LIN {X 0,Y 334.452,Z 401.269,A -85,B 0,C 180,E1 -14668.793,E2 -14668.793} C_VEL
LIN {X 0,Y 334.325,Z 404.538,A -85,B 0,C 180,E1 -14671.202,E2 -14671.202} C_VEL
LIN {X 0,Y 333.817,Z 411.373,A -85,B 0,C 180,E1 -14676.04,E2 -14676.04} C_VEL
LIN {X 0,Y 333.325,Z 416.707,A -85,B 0,C 180,E1 -14679.708,E2 -14679.708} C_VEL
LIN {X 0,Y 332.922,Z 422.789,A -85,B 0,C 180,E1 -14683.819,E2 -14683.819} C_VEL
LIN {X 0,Y 332.746,Z 425.377,A -85,B 0,C 180,E1 -14685.541,E2 -14685.541} C_VEL
LIN {X 0,Y 335.286,Z 437.671,A -85,B 0,C 180,E1 -14686.278,E2 -14686.278} C_VEL
LIN {X 0,Y 337.14,Z 448.371,A -85,B 0,C 180,E1 -14687.121,E2 -14687.121} C_VEL
LIN {X 0,Y 337.706,Z 453.161,A -85,B 0,C 180,E1 -14687.56,E2 -14687.56} C_VEL
LIN {X 0,Y 336.838,Z 463.101,A -85,B 0,C 180,E1 -14688.55,E2 -14688.55} C_VEL
LIN {X 0,Y 335.882,Z 473.522,A -85,B 0,C 180,E1 -14689.887,E2 -14689.887} C_VEL
LIN {X 0,Y 335.116,Z 481.598,A -85,B 0,C 180,E1 -14691.205,E2 -14691.205} C_VEL
LIN {X 0,Y 334.312,Z 488.548,A -85,B 0,C 180,E1 -14692.594,E2 -14692.594} C_VEL
LIN {X 0,Y 333.638,Z 495.183,A -85,B 0,C 180,E1 -14694.249,E2 -14694.249} C_VEL
LIN {X 0,Y 332.933,Z 501.458,A -85,B 0,C 180,E1 -14696.311,E2 -14696.311} C_VEL
LIN {X 0,Y 332.49,Z 505.928,A -85,B 0,C 180,E1 -14698.394,E2 -14698.394} C_VEL
LIN {X 0,Y 332.162,Z 508.838,A -85,B 0,C 180,E1 -14700.513,E2 -14700.513} C_VEL
LIN {X 0,Y 332.04,Z 510.039,A -85,B 0,C 180,E1 -14702.152,E2 -14702.152} C_VEL
LIN {X 0,Y 332.048,Z 510.377,A -85,B 0,C 180,E1 -14703.384,E2 -14703.384} C_VEL
LIN {X 0,Y 332.14,Z 510.099,A -85,B 0,C 180,E1 -14704.838,E2 -14704.838} C_VEL
LIN {X 0,Y 332.357,Z 508.921,A -85,B 0,C 180,E1 -14706.531,E2 -14706.531} C_VEL
LIN {X 0,Y 332.817,Z 506.101,A -85,B 0,C 180,E1 -14708.619,E2 -14708.619} C_VEL
LIN {X 0,Y 333.451,Z 501.852,A -85,B 0,C 180,E1 -14710.646,E2 -14710.646} C_VEL
LIN {X 0,Y 334.247,Z 496.051,A -85,B 0,C 180,E1 -14712.615,E2 -14712.615} C_VEL
LIN {X 0,Y 335.069,Z 490.017,A -85,B 0,C 180,E1 -14714.188,E2 -14714.188} C_VEL
LIN {X 0,Y 336.238,Z 481.51,A -85,B 0,C 180,E1 -14715.923,E2 -14715.923} C_VEL
LIN {X 0,Y 337.346,Z 473.22,A -85,B 0,C 180,E1 -14717.249,E2 -14717.249} C_VEL
LIN {X 0,Y 338.217,Z 465.547,A -85,B 0,C 180,E1 -14718.255,E2 -14718.255} C_VEL
LIN {X 0,Y 338.19,Z 462.356,A -85,B 0,C 180,E1 -14718.645,E2 -14718.645} C_VEL
LIN {X 0,Y 337.525,Z 459.239,A -85,B 0,C 180,E1 -14719.042,E2 -14719.042} C_VEL
LIN {X 0,Y 335.005,Z 453.218,A -85,B 0,C 180,E1 -14719.825,E2 -14719.825} C_VEL
LIN {X 0,Y 331.983,Z 447.052,A -85,B 0,C 180,E1 -14720.571,E2 -14720.571} C_VEL
LIN {X 0,Y 330.188,Z 442.057,A -85,B 0,C 180,E1 -14721.074,E2 -14721.074} C_VEL
LIN {X 0,Y 329.772,Z 440.283,A -85,B 0,C 180,E1 -14721.225,E2 -14721.225} C_VEL
LIN {X 0,Y 326.593,Z 428.367,A -85,B 0,C 180,E1 -14722.124,E2 -14722.124} C_VEL
LIN {X 0,Y 326.223,Z 426.561,A -85,B 0,C 180,E1 -14722.269,E2 -14722.269} C_VEL
LIN {X 0,Y 326.561,Z 421.444,A -85,B 0,C 180,E1 -14725.976,E2 -14725.976} C_VEL
LIN {X 0,Y 326.992,Z 415.563,A -85,B 0,C 180,E1 -14730.375,E2 -14730.375} C_VEL
LIN {X 0,Y 327.403,Z 411.837,A -85,B 0,C 180,E1 -14733.206,E2 -14733.206} C_VEL
LIN {X 0,Y 327.616,Z 408.363,A -85,B 0,C 180,E1 -14735.947,E2 -14735.947} C_VEL
LIN {X 0,Y 327.526,Z 405.191,A -85,B 0,C 180,E1 -14738.606,E2 -14738.606} C_VEL
LIN {X 0,Y 327.156,Z 402.286,A -85,B 0,C 180,E1 -14741.203,E2 -14741.203} C_VEL
LIN {X 0,Y 326.68,Z 399.798,A -85,B 0,C 180,E1 -14743.599,E2 -14743.599} C_VEL
LIN {X 0,Y 326.741,Z 399.788,A -85,B 0,C 180,E1 -14746.314,E2 -14746.314} C_VEL
LIN {X 0,Y 326.793,Z 399.779,A -85,B 0,C 180,E1 -14750.094,E2 -14750.094} C_VEL
LIN {X 0,Y 326.958,Z 399.76,A -85,B 0,C 180,E1 -14752.59,E2 -14752.59} C_VEL
LIN {X 0,Y 326.767,Z 399.785,A -85,B 0,C 180,E1 -14755.065,E2 -14755.065} C_VEL
LIN {X 0,Y 327.056,Z 399.748,A -85,B 0,C 180,E1 -14757.537,E2 -14757.537} C_VEL
LIN {X 0,Y 327.216,Z 399.727,A -85,B 0,C 180,E1 -14760,E2 -14760} C_VEL
LIN {X 0,Y 327.056,Z 399.747,A -85,B 0,C 180,E1 -14762.464,E2 -14762.464} C_VEL
LIN {X 0,Y 326.978,Z 399.751,A -85,B 0,C 180,E1 -14766.17,E2 -14766.17} C_VEL
LIN {X 0,Y 326.893,Z 399.765,A -85,B 0,C 180,E1 -14768.656,E2 -14768.656} C_VEL
LIN {X 0,Y 326.718,Z 399.783,A -85,B 0,C 180,E1 -14772.422,E2 -14772.422} C_VEL
LIN {X 0,Y 326.733,Z 399.783,A -85,B 0,C 180,E1 -14774.959,E2 -14774.959} C_VEL
LIN {X 0,Y 326.716,Z 399.783,A -85,B 0,C 180,E1 -14778.842,E2 -14778.842} C_VEL
LIN {X 0,Y 326.624,Z 399.801,A -85,B 0,C 180,E1 -14782.788,E2 -14782.788} C_VEL
LIN {X 0,Y 326.673,Z 399.794,A -85,B 0,C 180,E1 -14785.486,E2 -14785.486} C_VEL
LIN {X 0,Y 326.643,Z 399.792,A -85,B 0,C 180,E1 -14789.661,E2 -14789.661} C_VEL
LIN {X 0,Y 326.59,Z 399.804,A -85,B 0,C 180,E1 -14794.022,E2 -14794.022} C_VEL
LIN {X 0,Y 326.613,Z 399.802,A -85,B 0,C 180,E1 -14797.242,E2 -14797.242} C_VEL
LIN {X 0,Y 326.62,Z 399.801,A -85,B 0,C 180,E1 -14800.205,E2 -14800.205} C_VEL
LIN {X 0,Y 326.644,Z 399.799,A -85,B 0,C 180,E1 -14803.512,E2 -14803.512} C_VEL
LIN {X 0,Y 326.702,Z 399.906,A -85,B 0,C 180,E1 -14804.862,E2 -14804.862} C_VEL
LIN {X 0,Y 327.773,Z 405.318,A -85,B 0,C 180,E1 -14808.631,E2 -14808.631} C_VEL
LIN {X 0,Y 328.717,Z 410.195,A -85,B 0,C 180,E1 -14811.687,E2 -14811.687} C_VEL
LIN {X 0,Y 330.049,Z 416.95,A -85,B 0,C 180,E1 -14815.573,E2 -14815.573} C_VEL
LIN {X 0,Y 330.66,Z 421.324,A -85,B 0,C 180,E1 -14817.907,E2 -14817.907} C_VEL
LIN {X 0,Y 329.991,Z 425.615,A -85,B 0,C 180,E1 -14819.971,E2 -14819.971} C_VEL
LIN {X 0,Y 328.501,Z 434.354,A -85,B 0,C 180,E1 -14823.969,E2 -14823.969} C_VEL
LIN {X 0,Y 327.223,Z 443.457,A -85,B 0,C 180,E1 -14827.993,E2 -14827.993} C_VEL
LIN {X 0,Y 330.129,Z 458.426,A -85,B 0,C 180,E1 -14828.837,E2 -14828.837} C_VEL
LIN {X 0,Y 331.601,Z 471.167,A -85,B 0,C 180,E1 -14829.742,E2 -14829.742} C_VEL
LIN {X 0,Y 332.114,Z 482.072,A -85,B 0,C 180,E1 -14830.695,E2 -14830.695} C_VEL
LIN {X 0,Y 331.005,Z 492.541,A -85,B 0,C 180,E1 -14831.753,E2 -14831.753} C_VEL
LIN {X 0,Y 329.552,Z 503.242,A -85,B 0,C 180,E1 -14833.111,E2 -14833.111} C_VEL
LIN {X 0,Y 328.483,Z 512.049,A -85,B 0,C 180,E1 -14834.507,E2 -14834.507} C_VEL
LIN {X 0,Y 327.513,Z 519.964,A -85,B 0,C 180,E1 -14836.033,E2 -14836.033} C_VEL
LIN {X 0,Y 326.413,Z 527.732,A -85,B 0,C 180,E1 -14837.885,E2 -14837.885} C_VEL
LIN {X 0,Y 325.459,Z 536.929,A -85,B 0,C 180,E1 -14840.683,E2 -14840.683} C_VEL
LIN {X 0,Y 325.106,Z 542.054,A -85,B 0,C 180,E1 -14842.55,E2 -14842.55} C_VEL
LIN {X 0,Y 324.911,Z 545.74,A -85,B 0,C 180,E1 -14844.274,E2 -14844.274} C_VEL
LIN {X 0,Y 324.917,Z 548.848,A -85,B 0,C 180,E1 -14846.282,E2 -14846.282} C_VEL
LIN {X 0,Y 324.882,Z 550.174,A -85,B 0,C 180,E1 -14847.523,E2 -14847.523} C_VEL
LIN {X 0,Y 324.897,Z 551.09,A -85,B 0,C 180,E1 -14848.763,E2 -14848.763} C_VEL
LIN {X 0,Y 324.91,Z 551.588,A -85,B 0,C 180,E1 -14850.003,E2 -14850.003} C_VEL
LIN {X 0,Y 324.885,Z 551.632,A -85,B 0,C 180,E1 -14851.242,E2 -14851.242} C_VEL
LIN {X 0,Y 324.884,Z 551.275,A -85,B 0,C 180,E1 -14852.482,E2 -14852.482} C_VEL
LIN {X 0,Y 324.917,Z 550.521,A -85,B 0,C 180,E1 -14853.723,E2 -14853.723} C_VEL
LIN {X 0,Y 324.92,Z 548.385,A -85,B 0,C 180,E1 -14855.741,E2 -14855.741} C_VEL
LIN {X 0,Y 325.191,Z 545.655,A -85,B 0,C 180,E1 -14857.453,E2 -14857.453} C_VEL
LIN {X 0,Y 325.607,Z 541.696,A -85,B 0,C 180,E1 -14859.319,E2 -14859.319} C_VEL
LIN {X 0,Y 326.431,Z 535.61,A -85,B 0,C 180,E1 -14861.49,E2 -14861.49} C_VEL
LIN {X 0,Y 327.445,Z 528.982,A -85,B 0,C 180,E1 -14863.342,E2 -14863.342} C_VEL
LIN {X 0,Y 328.79,Z 520.814,A -85,B 0,C 180,E1 -14865.182,E2 -14865.182} C_VEL
LIN {X 0,Y 329.975,Z 512.524,A -85,B 0,C 180,E1 -14866.712,E2 -14866.712} C_VEL
LIN {X 0,Y 331.648,Z 502.355,A -85,B 0,C 180,E1 -14868.216,E2 -14868.216} C_VEL
LIN {X 0,Y 333.175,Z 492.443,A -85,B 0,C 180,E1 -14869.407,E2 -14869.407} C_VEL
LIN {X 0,Y 334.141,Z 483.521,A -85,B 0,C 180,E1 -14870.309,E2 -14870.309} C_VEL
LIN {X 0,Y 333.854,Z 472.11,A -85,B 0,C 180,E1 -14871.365,E2 -14871.365} C_VEL
LIN {X 0,Y 332.316,Z 458.96,A -85,B 0,C 180,E1 -14872.419,E2 -14872.419} C_VEL
LIN {X 0,Y 329.655,Z 445.962,A -85,B 0,C 180,E1 -14873.306,E2 -14873.306} C_VEL
LIN {X 0,Y 327.517,Z 437.12,A -85,B 0,C 180,E1 -14873.863,E2 -14873.863} C_VEL
LIN {X 0,Y 328.673,Z 429.043,A -85,B 0,C 180,E1 -14877.372,E2 -14877.372} C_VEL
LIN {X 0,Y 329.908,Z 421.406,A -85,B 0,C 180,E1 -14880.751,E2 -14880.751} C_VEL
LIN {X 0,Y 330.137,Z 418.339,A -85,B 0,C 180,E1 -14882.157,E2 -14882.157} C_VEL
LIN {X 0,Y 329.022,Z 412.165,A -85,B 0,C 180,E1 -14885.223,E2 -14885.223} C_VEL
LIN {X 0,Y 327.48,Z 404.167,A -85,B 0,C 180,E1 -14889.412,E2 -14889.412} C_VEL
LIN {X 0,Y 326.602,Z 399.803,A -85,B 0,C 180,E1 -14891.844,E2 -14891.844} C_VEL
LIN {X 0,Y 326.532,Z 399.81,A -85,B 0,C 180,E1 -14895.259,E2 -14895.259} C_VEL
LIN {X 0,Y 326.569,Z 399.805,A -85,B 0,C 180,E1 -14898.153,E2 -14898.153} C_VEL
LIN {X 0,Y 326.59,Z 399.798,A -85,B 0,C 180,E1 -14901.386,E2 -14901.386} C_VEL
LIN {X 0,Y 326.627,Z 399.8,A -85,B 0,C 180,E1 -14904.852,E2 -14904.852} C_VEL
LIN {X 0,Y 326.616,Z 399.8,A -85,B 0,C 180,E1 -14907.456,E2 -14907.456} C_VEL
LIN {X 0,Y 326.597,Z 399.802,A -85,B 0,C 180,E1 -14910.334,E2 -14910.334} C_VEL
LIN {X 0,Y 326.603,Z 399.802,A -85,B 0,C 180,E1 -14913.135,E2 -14913.135} C_VEL
LIN {X 0,Y 326.598,Z 399.803,A -85,B 0,C 180,E1 -14917.211,E2 -14917.211} C_VEL
LIN {X 0,Y 326.754,Z 399.784,A -85,B 0,C 180,E1 -14921.178,E2 -14921.178} C_VEL
LIN {X 0,Y 326.772,Z 399.784,A -85,B 0,C 180,E1 -14925.433,E2 -14925.433} C_VEL
LIN {X 0,Y 326.788,Z 399.871,A -85,B 0,C 180,E1 -14929.545,E2 -14929.545} C_VEL
LIN {X 0,Y 327.805,Z 404.409,A -85,B 0,C 180,E1 -14932.609,E2 -14932.609} C_VEL
LIN {X 0,Y 328.363,Z 408.303,A -85,B 0,C 180,E1 -14935.088,E2 -14935.088} C_VEL
LIN {X 0,Y 328.368,Z 412.44,A -85,B 0,C 180,E1 -14937.546,E2 -14937.546} C_VEL
LIN {X 0,Y 327.807,Z 417.739,A -85,B 0,C 180,E1 -14940.614,E2 -14940.614} C_VEL
LIN {X 0,Y 327.262,Z 425.21,A -85,B 0,C 180,E1 -14944.927,E2 -14944.927} C_VEL
LIN {X 0,Y 327.074,Z 428.969,A -85,B 0,C 180,E1 -14947.097,E2 -14947.097} C_VEL
LIN {X 0,Y 331.673,Z 443.489,A -85,B 0,C 180,E1 -14948.319,E2 -14948.319} C_VEL
LIN {X 0,Y 334.363,Z 455.286,A -85,B 0,C 180,E1 -14949.406,E2 -14949.406} C_VEL
LIN {X 0,Y 335.716,Z 465.144,A -85,B 0,C 180,E1 -14950.402,E2 -14950.402} C_VEL
LIN {X 0,Y 334.254,Z 476.454,A -85,B 0,C 180,E1 -14951.522,E2 -14951.522} C_VEL
LIN {X 0,Y 332.591,Z 487.852,A -85,B 0,C 180,E1 -14952.949,E2 -14952.949} C_VEL
LIN {X 0,Y 331.025,Z 497.442,A -85,B 0,C 180,E1 -14954.445,E2 -14954.445} C_VEL
LIN {X 0,Y 329.425,Z 506.719,A -85,B 0,C 180,E1 -14956.248,E2 -14956.248} C_VEL
LIN {X 0,Y 328.113,Z 514.369,A -85,B 0,C 180,E1 -14958.094,E2 -14958.094} C_VEL
LIN {X 0,Y 326.984,Z 520.949,A -85,B 0,C 180,E1 -14960.114,E2 -14960.114} C_VEL
LIN {X 0,Y 326.086,Z 525.896,A -85,B 0,C 180,E1 -14962.061,E2 -14962.061} C_VEL
LIN {X 0,Y 325.474,Z 529.964,A -85,B 0,C 180,E1 -14964.221,E2 -14964.221} C_VEL
LIN {X 0,Y 325.17,Z 531.838,A -85,B 0,C 180,E1 -14965.611,E2 -14965.611} C_VEL
LIN {X 0,Y 324.841,Z 533.562,A -85,B 0,C 180,E1 -14967.493,E2 -14967.493} C_VEL
LIN {X 0,Y 324.622,Z 534.411,A -85,B 0,C 180,E1 -14970.001,E2 -14970.001} C_VEL
LIN {X 0,Y 324.582,Z 533.648,A -85,B 0,C 180,E1 -14972.385,E2 -14972.385} C_VEL
LIN {X 0,Y 324.76,Z 531.489,A -85,B 0,C 180,E1 -14974.677,E2 -14974.677} C_VEL
LIN {X 0,Y 325.157,Z 528.008,A -85,B 0,C 180,E1 -14976.894,E2 -14976.894} C_VEL
LIN {X 0,Y 325.542,Z 523.285,A -85,B 0,C 180,E1 -14978.993,E2 -14978.993} C_VEL
LIN {X 0,Y 326.14,Z 517.232,A -85,B 0,C 180,E1 -14981.041,E2 -14981.041} C_VEL
LIN {X 0,Y 326.915,Z 509.69,A -85,B 0,C 180,E1 -14983.033,E2 -14983.033} C_VEL
LIN {X 0,Y 327.913,Z 500.349,A -85,B 0,C 180,E1 -14984.984,E2 -14984.984} C_VEL
LIN {X 0,Y 329.014,Z 490.812,A -85,B 0,C 180,E1 -14986.574,E2 -14986.574} C_VEL
LIN {X 0,Y 330.099,Z 480.41,A -85,B 0,C 180,E1 -14987.98,E2 -14987.98} C_VEL
LIN {X 0,Y 331.204,Z 469.031,A -85,B 0,C 180,E1 -14989.216,E2 -14989.216} C_VEL
LIN {X 0,Y 331.864,Z 460.882,A -85,B 0,C 180,E1 -14989.933,E2 -14989.933} C_VEL
LIN {X 0,Y 330.017,Z 448.543,A -85,B 0,C 180,E1 -14990.934,E2 -14990.934} C_VEL
LIN {X 0,Y 327.287,Z 434.324,A -85,B 0,C 180,E1 -14991.825,E2 -14991.825} C_VEL
LIN {X 0,Y 325.942,Z 427.724,A -85,B 0,C 180,E1 -14992.178,E2 -14992.178} C_VEL
LIN {X 0,Y 326.253,Z 420.978,A -85,B 0,C 180,E1 -14995.936,E2 -14995.936} C_VEL
LIN {X 0,Y 326.542,Z 414.759,A -85,B 0,C 180,E1 -14999.417,E2 -14999.417} C_VEL
LIN {X 0,Y 326.776,Z 409.236,A -85,B 0,C 180,E1 -15002.507,E2 -15002.507} C_VEL
LIN {X 0,Y 327.051,Z 403.236,A -85,B 0,C 180,E1 -15005.9,E2 -15005.9} C_VEL
LIN {X 0,Y 326.775,Z 399.782,A -85,B 0,C 180,E1 -15007.93,E2 -15007.93} C_VEL
LIN {X 0,Y 326.747,Z 399.785,A -85,B 0,C 180,E1 -15011.175,E2 -15011.175} C_VEL
LIN {X 0,Y 326.765,Z 399.784,A -85,B 0,C 180,E1 -15015.431,E2 -15015.431} C_VEL
LIN {X 0,Y 326.771,Z 399.782,A -85,B 0,C 180,E1 -15018.836,E2 -15018.836} C_VEL
LIN {X 0,Y 326.923,Z 399.764,A -85,B 0,C 180,E1 -15022.587,E2 -15022.587} C_VEL
LIN {X 0,Y 326.754,Z 399.789,A -85,B 0,C 180,E1 -15025.062,E2 -15025.062} C_VEL
LIN {X 0,Y 326.832,Z 399.839,A -85,B 0,C 180,E1 -15026.761,E2 -15026.761} C_VEL
LIN {X 0,Y 327.447,Z 402.365,A -85,B 0,C 180,E1 -15028.767,E2 -15028.767} C_VEL
LIN {X 0,Y 327.295,Z 405.666,A -85,B 0,C 180,E1 -15031.228,E2 -15031.228} C_VEL
LIN {X 0,Y 326.744,Z 412.542,A -85,B 0,C 180,E1 -15036.171,E2 -15036.171} C_VEL
LIN {X 0,Y 326.262,Z 417.889,A -85,B 0,C 180,E1 -15039.92,E2 -15039.92} C_VEL
LIN {X 0,Y 325.847,Z 423.753,A -85,B 0,C 180,E1 -15043.935,E2 -15043.935} C_VEL
LIN {X 0,Y 325.743,Z 425.557,A -85,B 0,C 180,E1 -15045.162,E2 -15045.162} C_VEL
LIN {X 0,Y 328.436,Z 438.699,A -85,B 0,C 180,E1 -15045.989,E2 -15045.989} C_VEL
LIN {X 0,Y 330.221,Z 449.282,A -85,B 0,C 180,E1 -15046.853,E2 -15046.853} C_VEL
LIN {X 0,Y 330.806,Z 453.971,A -85,B 0,C 180,E1 -15047.3,E2 -15047.3} C_VEL
LIN {X 0,Y 329.915,Z 463.778,A -85,B 0,C 180,E1 -15048.31,E2 -15048.31} C_VEL
LIN {X 0,Y 328.986,Z 473.555,A -85,B 0,C 180,E1 -15049.59,E2 -15049.59} C_VEL
LIN {X 0,Y 328.119,Z 482.163,A -85,B 0,C 180,E1 -15051.021,E2 -15051.021} C_VEL
LIN {X 0,Y 327.137,Z 490.412,A -85,B 0,C 180,E1 -15052.746,E2 -15052.746} C_VEL
LIN {X 0,Y 326.37,Z 497.455,A -85,B 0,C 180,E1 -15054.663,E2 -15054.663} C_VEL
LIN {X 0,Y 325.87,Z 501.929,A -85,B 0,C 180,E1 -15056.236,E2 -15056.236} C_VEL
LIN {X 0,Y 325.414,Z 506.379,A -85,B 0,C 180,E1 -15058.364,E2 -15058.364} C_VEL
LIN {X 0,Y 325.128,Z 508.903,A -85,B 0,C 180,E1 -15060.159,E2 -15060.159} C_VEL
LIN {X 0,Y 325.001,Z 509.9,A -85,B 0,C 180,E1 -15061.26,E2 -15061.26} C_VEL
LIN {X 0,Y 324.963,Z 510.663,A -85,B 0,C 180,E1 -15062.726,E2 -15062.726} C_VEL
LIN {X 0,Y 325.051,Z 510.568,A -85,B 0,C 180,E1 -15064.755,E2 -15064.755} C_VEL
LIN {X 0,Y 325.356,Z 509.042,A -85,B 0,C 180,E1 -15066.944,E2 -15066.944} C_VEL
LIN {X 0,Y 325.893,Z 506.035,A -85,B 0,C 180,E1 -15069.073,E2 -15069.073} C_VEL
LIN {X 0,Y 326.539,Z 501.602,A -85,B 0,C 180,E1 -15071.124,E2 -15071.124} C_VEL
LIN {X 0,Y 327.443,Z 495.596,A -85,B 0,C 180,E1 -15073.135,E2 -15073.135} C_VEL
LIN {X 0,Y 328.451,Z 488.585,A -85,B 0,C 180,E1 -15074.914,E2 -15074.914} C_VEL
LIN {X 0,Y 329.56,Z 480.771,A -85,B 0,C 180,E1 -15076.469,E2 -15076.469} C_VEL
LIN {X 0,Y 330.919,Z 470.893,A -85,B 0,C 180,E1 -15078.01,E2 -15078.01} C_VEL
LIN {X 0,Y 332.054,Z 461.076,A -85,B 0,C 180,E1 -15079.202,E2 -15079.202} C_VEL
LIN {X 0,Y 332.497,Z 456.981,A -85,B 0,C 180,E1 -15079.619,E2 -15079.619} C_VEL
LIN {X 0,Y 331.184,Z 447.065,A -85,B 0,C 180,E1 -15080.627,E2 -15080.627} C_VEL
LIN {X 0,Y 329.772,Z 440.283,A -85,B 0,C 180,E1 -15081.225,E2 -15081.225} C_VEL
LIN {X 0,Y 328.516,Z 438.347,A -85,B 0,C 180,E1 -15081.451,E2 -15081.451} C_VEL
LIN {X 0,Y 322.469,Z 435.25,A -85,B 0,C 180,E1 -15082.111,E2 -15082.111} C_VEL
LIN {X 0,Y 321.128,Z 433.6,A -85,B 0,C 180,E1 -15082.304,E2 -15082.304} C_VEL
LIN {X 0,Y 319.257,Z 426.842,A -85,B 0,C 180,E1 -15082.787,E2 -15082.787} C_VEL
LIN {X 0,Y 319.608,Z 421.628,A -85,B 0,C 180,E1 -15086.671,E2 -15086.671} C_VEL
LIN {X 0,Y 319.882,Z 417.736,A -85,B 0,C 180,E1 -15089.648,E2 -15089.648} C_VEL
LIN {X 0,Y 320.324,Z 413.962,A -85,B 0,C 180,E1 -15092.565,E2 -15092.565} C_VEL
LIN {X 0,Y 320.608,Z 410.436,A -85,B 0,C 180,E1 -15095.387,E2 -15095.387} C_VEL
LIN {X 0,Y 320.602,Z 407.183,A -85,B 0,C 180,E1 -15098.121,E2 -15098.121} C_VEL
LIN {X 0,Y 320.283,Z 404.248,A -85,B 0,C 180,E1 -15100.783,E2 -15100.783} C_VEL
LIN {X 0,Y 319.672,Z 400.67,A -85,B 0,C 180,E1 -15104.377,E2 -15104.377} C_VEL
LIN {X 0,Y 319.664,Z 400.667,A -85,B 0,C 180,E1 -15107.3,E2 -15107.3} C_VEL
LIN {X 0,Y 319.859,Z 400.644,A -85,B 0,C 180,E1 -15111.369,E2 -15111.369} C_VEL
LIN {X 0,Y 319.932,Z 400.633,A -85,B 0,C 180,E1 -15113.695,E2 -15113.695} C_VEL
LIN {X 0,Y 319.996,Z 400.627,A -85,B 0,C 180,E1 -15117.483,E2 -15117.483} C_VEL
LIN {X 0,Y 320.167,Z 400.605,A -85,B 0,C 180,E1 -15120,E2 -15120} C_VEL
LIN {X 0,Y 319.996,Z 400.626,A -85,B 0,C 180,E1 -15122.518,E2 -15122.518} C_VEL
LIN {X 0,Y 319.933,Z 400.628,A -85,B 0,C 180,E1 -15126.306,E2 -15126.306} C_VEL
LIN {X 0,Y 319.821,Z 400.645,A -85,B 0,C 180,E1 -15128.849,E2 -15128.849} C_VEL
LIN {X 0,Y 319.664,Z 400.661,A -85,B 0,C 180,E1 -15132.701,E2 -15132.701} C_VEL
LIN {X 0,Y 319.679,Z 400.66,A -85,B 0,C 180,E1 -15135.297,E2 -15135.297} C_VEL
LIN {X 0,Y 319.66,Z 400.664,A -85,B 0,C 180,E1 -15139.256,E2 -15139.256} C_VEL
LIN {X 0,Y 319.566,Z 400.679,A -85,B 0,C 180,E1 -15143.32,E2 -15143.32} C_VEL
LIN {X 0,Y 319.617,Z 400.672,A -85,B 0,C 180,E1 -15146.09,E2 -15146.09} C_VEL
LIN {X 0,Y 319.571,Z 400.676,A -85,B 0,C 180,E1 -15148.936,E2 -15148.936} C_VEL
LIN {X 0,Y 319.515,Z 400.681,A -85,B 0,C 180,E1 -15151.864,E2 -15151.864} C_VEL
LIN {X 0,Y 319.563,Z 400.679,A -85,B 0,C 180,E1 -15155.546,E2 -15155.546} C_VEL
LIN {X 0,Y 319.584,Z 400.677,A -85,B 0,C 180,E1 -15158.007,E2 -15158.007} C_VEL
LIN {X 0,Y 319.587,Z 400.678,A -85,B 0,C 180,E1 -15161.615,E2 -15161.615} C_VEL
LIN {X 0,Y 319.629,Z 400.846,A -85,B 0,C 180,E1 -15164.042,E2 -15164.042} C_VEL
LIN {X 0,Y 320.545,Z 405.112,A -85,B 0,C 180,E1 -15167.187,E2 -15167.187} C_VEL
LIN {X 0,Y 321.557,Z 410.35,A -85,B 0,C 180,E1 -15170.672,E2 -15170.672} C_VEL
LIN {X 0,Y 322.851,Z 417.144,A -85,B 0,C 180,E1 -15174.774,E2 -15174.774} C_VEL
LIN {X 0,Y 323.599,Z 421.346,A -85,B 0,C 180,E1 -15177.119,E2 -15177.119} C_VEL
LIN {X 0,Y 323.545,Z 424.16,A -85,B 0,C 180,E1 -15178.583,E2 -15178.583} C_VEL
LIN {X 0,Y 321.886,Z 432.837,A -85,B 0,C 180,E1 -15182.713,E2 -15182.713} C_VEL
LIN {X 0,Y 320.53,Z 441.69,A -85,B 0,C 180,E1 -15186.758,E2 -15186.758} C_VEL
LIN {X 0,Y 320.32,Z 443.398,A -85,B 0,C 180,E1 -15187.485,E2 -15187.485} C_VEL
LIN {X 0,Y 322.976,Z 456.392,A -85,B 0,C 180,E1 -15188.214,E2 -15188.214} C_VEL
LIN {X 0,Y 324.618,Z 468.94,A -85,B 0,C 180,E1 -15189.111,E2 -15189.111} C_VEL
LIN {X 0,Y 325.293,Z 480.354,A -85,B 0,C 180,E1 -15190.109,E2 -15190.109} C_VEL
LIN {X 0,Y 325.034,Z 486.85,A -85,B 0,C 180,E1 -15190.75,E2 -15190.75} C_VEL
LIN {X 0,Y 323.571,Z 497.51,A -85,B 0,C 180,E1 -15191.974,E2 -15191.974} C_VEL
LIN {X 0,Y 322.031,Z 508.166,A -85,B 0,C 180,E1 -15193.521,E2 -15193.521} C_VEL
LIN {X 0,Y 320.935,Z 516.769,A -85,B 0,C 180,E1 -15195.093,E2 -15195.093} C_VEL
LIN {X 0,Y 319.848,Z 525.08,A -85,B 0,C 180,E1 -15196.987,E2 -15196.987} C_VEL
LIN {X 0,Y 318.966,Z 530.728,A -85,B 0,C 180,E1 -15198.565,E2 -15198.565} C_VEL
LIN {X 0,Y 318.154,Z 539.994,A -85,B 0,C 180,E1 -15201.748,E2 -15201.748} C_VEL
LIN {X 0,Y 317.889,Z 544.379,A -85,B 0,C 180,E1 -15203.656,E2 -15203.656} C_VEL
LIN {X 0,Y 317.814,Z 546.681,A -85,B 0,C 180,E1 -15204.928,E2 -15204.928} C_VEL
LIN {X 0,Y 317.823,Z 548.525,A -85,B 0,C 180,E1 -15206.199,E2 -15206.199} C_VEL
LIN {X 0,Y 317.801,Z 549.88,A -85,B 0,C 180,E1 -15207.468,E2 -15207.468} C_VEL
LIN {X 0,Y 317.805,Z 550.824,A -85,B 0,C 180,E1 -15208.736,E2 -15208.736} C_VEL
LIN {X 0,Y 317.816,Z 551.364,A -85,B 0,C 180,E1 -15210.003,E2 -15210.003} C_VEL
LIN {X 0,Y 317.794,Z 551.45,A -85,B 0,C 180,E1 -15211.27,E2 -15211.27} C_VEL
LIN {X 0,Y 317.802,Z 551.12,A -85,B 0,C 180,E1 -15212.538,E2 -15212.538} C_VEL
LIN {X 0,Y 317.823,Z 550.391,A -85,B 0,C 180,E1 -15213.806,E2 -15213.806} C_VEL
LIN {X 0,Y 317.838,Z 548.503,A -85,B 0,C 180,E1 -15215.707,E2 -15215.707} C_VEL
LIN {X 0,Y 318.13,Z 545.63,A -85,B 0,C 180,E1 -15217.62,E2 -15217.62} C_VEL
LIN {X 0,Y 318.588,Z 541.745,A -85,B 0,C 180,E1 -15219.526,E2 -15219.526} C_VEL
LIN {X 0,Y 319.321,Z 536.731,A -85,B 0,C 180,E1 -15221.427,E2 -15221.427} C_VEL
LIN {X 0,Y 320.305,Z 530.452,A -85,B 0,C 180,E1 -15223.322,E2 -15223.322} C_VEL
LIN {X 0,Y 321.718,Z 522.637,A -85,B 0,C 180,E1 -15225.2,E2 -15225.2} C_VEL
LIN {X 0,Y 323.194,Z 512.985,A -85,B 0,C 180,E1 -15227.073,E2 -15227.073} C_VEL
LIN {X 0,Y 324.951,Z 503.049,A -85,B 0,C 180,E1 -15228.606,E2 -15228.606} C_VEL
LIN {X 0,Y 326.55,Z 493.382,A -85,B 0,C 180,E1 -15229.817,E2 -15229.817} C_VEL
LIN {X 0,Y 327.62,Z 484.775,A -85,B 0,C 180,E1 -15230.732,E2 -15230.732} C_VEL
LIN {X 0,Y 327.406,Z 473.351,A -85,B 0,C 180,E1 -15231.84,E2 -15231.84} C_VEL
LIN {X 0,Y 326.036,Z 460.605,A -85,B 0,C 180,E1 -15232.917,E2 -15232.917} C_VEL
LIN {X 0,Y 323.471,Z 447.178,A -85,B 0,C 180,E1 -15233.903,E2 -15233.903} C_VEL
LIN {X 0,Y 320.742,Z 436.804,A -85,B 0,C 180,E1 -15234.605,E2 -15234.605} C_VEL
LIN {X 0,Y 320.705,Z 436.092,A -85,B 0,C 180,E1 -15234.694,E2 -15234.694} C_VEL
LIN {X 0,Y 322.082,Z 427.151,A -85,B 0,C 180,E1 -15238.691,E2 -15238.691} C_VEL
LIN {X 0,Y 323.061,Z 421.055,A -85,B 0,C 180,E1 -15241.476,E2 -15241.476} C_VEL
LIN {X 0,Y 322.908,Z 417.996,A -85,B 0,C 180,E1 -15242.967,E2 -15242.967} C_VEL
LIN {X 0,Y 321.703,Z 411.78,A -85,B 0,C 180,E1 -15246.149,E2 -15246.149} C_VEL
LIN {X 0,Y 320.405,Z 404.942,A -85,B 0,C 180,E1 -15249.85,E2 -15249.85} C_VEL
LIN {X 0,Y 319.543,Z 400.684,A -85,B 0,C 180,E1 -15252.347,E2 -15252.347} C_VEL
LIN {X 0,Y 319.526,Z 400.677,A -85,B 0,C 180,E1 -15256.541,E2 -15256.541} C_VEL
LIN {X 0,Y 319.553,Z 400.679,A -85,B 0,C 180,E1 -15260.371,E2 -15260.371} C_VEL
LIN {X 0,Y 319.587,Z 400.675,A -85,B 0,C 180,E1 -15264.458,E2 -15264.458} C_VEL
LIN {X 0,Y 319.532,Z 400.684,A -85,B 0,C 180,E1 -15268.138,E2 -15268.138} C_VEL
LIN {X 0,Y 319.575,Z 400.678,A -85,B 0,C 180,E1 -15271.606,E2 -15271.606} C_VEL
LIN {X 0,Y 319.534,Z 400.685,A -85,B 0,C 180,E1 -15275.298,E2 -15275.298} C_VEL
LIN {X 0,Y 319.573,Z 400.679,A -85,B 0,C 180,E1 -15278.046,E2 -15278.046} C_VEL
LIN {X 0,Y 319.698,Z 400.663,A -85,B 0,C 180,E1 -15280.963,E2 -15280.963} C_VEL
LIN {X 0,Y 319.74,Z 400.661,A -85,B 0,C 180,E1 -15285.276,E2 -15285.276} C_VEL
LIN {X 0,Y 319.721,Z 400.777,A -85,B 0,C 180,E1 -15288.589,E2 -15288.589} C_VEL
LIN {X 0,Y 320.589,Z 404.376,A -85,B 0,C 180,E1 -15291.172,E2 -15291.172} C_VEL
LIN {X 0,Y 321.305,Z 408.134,A -85,B 0,C 180,E1 -15293.721,E2 -15293.721} C_VEL
LIN {X 0,Y 321.59,Z 412.111,A -85,B 0,C 180,E1 -15296.24,E2 -15296.24} C_VEL
LIN {X 0,Y 321.307,Z 416.287,A -85,B 0,C 180,E1 -15298.746,E2 -15298.746} C_VEL
LIN {X 0,Y 320.454,Z 424.812,A -85,B 0,C 180,E1 -15303.772,E2 -15303.772} C_VEL
LIN {X 0,Y 320.229,Z 429.416,A -85,B 0,C 180,E1 -15306.379,E2 -15306.379} C_VEL
LIN {X 0,Y 324.781,Z 443.108,A -85,B 0,C 180,E1 -15307.589,E2 -15307.589} C_VEL
LIN {X 0,Y 327.728,Z 455.554,A -85,B 0,C 180,E1 -15308.788,E2 -15308.788} C_VEL
LIN {X 0,Y 329.115,Z 465.432,A -85,B 0,C 180,E1 -15309.836,E2 -15309.836} C_VEL
LIN {X 0,Y 328.513,Z 471.861,A -85,B 0,C 180,E1 -15310.476,E2 -15310.476} C_VEL
LIN {X 0,Y 326.819,Z 483.251,A -85,B 0,C 180,E1 -15311.788,E2 -15311.788} C_VEL
LIN {X 0,Y 325.063,Z 494.055,A -85,B 0,C 180,E1 -15313.359,E2 -15313.359} C_VEL
LIN {X 0,Y 323.281,Z 503.738,A -85,B 0,C 180,E1 -15315.122,E2 -15315.122} C_VEL
LIN {X 0,Y 321.98,Z 511.203,A -85,B 0,C 180,E1 -15316.81,E2 -15316.81} C_VEL
LIN {X 0,Y 320.574,Z 518.488,A -85,B 0,C 180,E1 -15318.866,E2 -15318.866} C_VEL
LIN {X 0,Y 319.676,Z 523.384,A -85,B 0,C 180,E1 -15320.594,E2 -15320.594} C_VEL
LIN {X 0,Y 318.789,Z 528.137,A -85,B 0,C 180,E1 -15322.763,E2 -15322.763} C_VEL
LIN {X 0,Y 318.202,Z 531.736,A -85,B 0,C 180,E1 -15325.099,E2 -15325.099} C_VEL
LIN {X 0,Y 317.941,Z 532.939,A -85,B 0,C 180,E1 -15326.237,E2 -15326.237} C_VEL
LIN {X 0,Y 317.7,Z 534.043,A -85,B 0,C 180,E1 -15327.762,E2 -15327.762} C_VEL
LIN {X 0,Y 317.555,Z 534.542,A -85,B 0,C 180,E1 -15329.136,E2 -15329.136} C_VEL
LIN {X 0,Y 317.489,Z 534.526,A -85,B 0,C 180,E1 -15330.606,E2 -15330.606} C_VEL
LIN {X 0,Y 317.498,Z 533.561,A -85,B 0,C 180,E1 -15332.735,E2 -15332.735} C_VEL
LIN {X 0,Y 317.741,Z 531.109,A -85,B 0,C 180,E1 -15335.105,E2 -15335.105} C_VEL
LIN {X 0,Y 318.16,Z 527.406,A -85,B 0,C 180,E1 -15337.321,E2 -15337.321} C_VEL
LIN {X 0,Y 318.548,Z 522.498,A -85,B 0,C 180,E1 -15339.446,E2 -15339.446} C_VEL
LIN {X 0,Y 319.176,Z 516.195,A -85,B 0,C 180,E1 -15341.523,E2 -15341.523} C_VEL
LIN {X 0,Y 320.083,Z 508.286,A -85,B 0,C 180,E1 -15343.564,E2 -15343.564} C_VEL
LIN {X 0,Y 321.005,Z 499.94,A -85,B 0,C 180,E1 -15345.298,E2 -15345.298} C_VEL
LIN {X 0,Y 322.149,Z 490.011,A -85,B 0,C 180,E1 -15346.956,E2 -15346.956} C_VEL
LIN {X 0,Y 323.258,Z 479.663,A -85,B 0,C 180,E1 -15348.361,E2 -15348.361} C_VEL
LIN {X 0,Y 324.352,Z 468.9,A -85,B 0,C 180,E1 -15349.535,E2 -15349.535} C_VEL
LIN {X 0,Y 324.797,Z 460.112,A -85,B 0,C 180,E1 -15350.331,E2 -15350.331} C_VEL
LIN {X 0,Y 322.782,Z 447.753,A -85,B 0,C 180,E1 -15351.343,E2 -15351.343} C_VEL
LIN {X 0,Y 320.139,Z 433.816,A -85,B 0,C 180,E1 -15352.226,E2 -15352.226} C_VEL
LIN {X 0,Y 318.912,Z 427.849,A -85,B 0,C 180,E1 -15352.556,E2 -15352.556} C_VEL
LIN {X 0,Y 319.306,Z 420.661,A -85,B 0,C 180,E1 -15356.613,E2 -15356.613} C_VEL
LIN {X 0,Y 319.59,Z 414.061,A -85,B 0,C 180,E1 -15360.342,E2 -15360.342} C_VEL
LIN {X 0,Y 319.902,Z 407.206,A -85,B 0,C 180,E1 -15364.254,E2 -15364.254} C_VEL
LIN {X 0,Y 320.043,Z 402.912,A -85,B 0,C 180,E1 -15366.715,E2 -15366.715} C_VEL
LIN {X 0,Y 319.713,Z 400.662,A -85,B 0,C 180,E1 -15368.054,E2 -15368.054} C_VEL
LIN {X 0,Y 319.661,Z 400.669,A -85,B 0,C 180,E1 -15372.071,E2 -15372.071} C_VEL
LIN {X 0,Y 319.734,Z 400.658,A -85,B 0,C 180,E1 -15376.005,E2 -15376.005} C_VEL
LIN {X 0,Y 319.753,Z 400.658,A -85,B 0,C 180,E1 -15379.87,E2 -15379.87} C_VEL
LIN {X 0,Y 319.908,Z 400.64,A -85,B 0,C 180,E1 -15383.691,E2 -15383.691} C_VEL
LIN {X 0,Y 319.763,Z 400.738,A -85,B 0,C 180,E1 -15386.532,E2 -15386.532} C_VEL
LIN {X 0,Y 320.44,Z 403.46,A -85,B 0,C 180,E1 -15388.741,E2 -15388.741} C_VEL
LIN {X 0,Y 320.264,Z 406.784,A -85,B 0,C 180,E1 -15391.255,E2 -15391.255} C_VEL
LIN {X 0,Y 319.675,Z 413.698,A -85,B 0,C 180,E1 -15396.308,E2 -15396.308} C_VEL
LIN {X 0,Y 319.186,Z 419.089,A -85,B 0,C 180,E1 -15400.142,E2 -15400.142} C_VEL
LIN {X 0,Y 318.785,Z 424.754,A -85,B 0,C 180,E1 -15404.064,E2 -15404.064} C_VEL
LIN {X 0,Y 318.702,Z 425.83,A -85,B 0,C 180,E1 -15404.809,E2 -15404.809} C_VEL
LIN {X 0,Y 321.063,Z 436.996,A -85,B 0,C 180,E1 -15405.489,E2 -15405.489} C_VEL
LIN {X 0,Y 323.057,Z 448.564,A -85,B 0,C 180,E1 -15406.425,E2 -15406.425} C_VEL
LIN {X 0,Y 323.859,Z 455.789,A -85,B 0,C 180,E1 -15407.13,E2 -15407.13} C_VEL
LIN {X 0,Y 322.871,Z 465.871,A -85,B 0,C 180,E1 -15408.231,E2 -15408.231} C_VEL
LIN {X 0,Y 322.034,Z 474.219,A -85,B 0,C 180,E1 -15409.374,E2 -15409.374} C_VEL
LIN {X 0,Y 321.127,Z 482.729,A -85,B 0,C 180,E1 -15410.829,E2 -15410.829} C_VEL
LIN {X 0,Y 320.275,Z 489.791,A -85,B 0,C 180,E1 -15412.318,E2 -15412.318} C_VEL
LIN {X 0,Y 319.554,Z 496.172,A -85,B 0,C 180,E1 -15414.005,E2 -15414.005} C_VEL
LIN {X 0,Y 319.034,Z 500.486,A -85,B 0,C 180,E1 -15415.421,E2 -15415.421} C_VEL
LIN {X 0,Y 318.466,Z 505.54,A -85,B 0,C 180,E1 -15417.605,E2 -15417.605} C_VEL
LIN {X 0,Y 318.218,Z 507.951,A -85,B 0,C 180,E1 -15419.066,E2 -15419.066} C_VEL
LIN {X 0,Y 317.992,Z 509.699,A -85,B 0,C 180,E1 -15420.548,E2 -15420.548} C_VEL
LIN {X 0,Y 317.871,Z 511.085,A -85,B 0,C 180,E1 -15422.843,E2 -15422.843} C_VEL
LIN {X 0,Y 318.031,Z 510.875,A -85,B 0,C 180,E1 -15425.151,E2 -15425.151} C_VEL
LIN {X 0,Y 318.363,Z 509.139,A -85,B 0,C 180,E1 -15427.372,E2 -15427.372} C_VEL
LIN {X 0,Y 318.944,Z 505.978,A -85,B 0,C 180,E1 -15429.536,E2 -15429.536} C_VEL
LIN {X 0,Y 319.688,Z 501.352,A -85,B 0,C 180,E1 -15431.63,E2 -15431.63} C_VEL
LIN {X 0,Y 320.663,Z 495.124,A -85,B 0,C 180,E1 -15433.676,E2 -15433.676} C_VEL
LIN {X 0,Y 321.612,Z 488.97,A -85,B 0,C 180,E1 -15435.246,E2 -15435.246} C_VEL
LIN {X 0,Y 322.779,Z 481.161,A -85,B 0,C 180,E1 -15436.831,E2 -15436.831} C_VEL
LIN {X 0,Y 324.117,Z 471.855,A -85,B 0,C 180,E1 -15438.325,E2 -15438.325} C_VEL
LIN {X 0,Y 325.391,Z 461.53,A -85,B 0,C 180,E1 -15439.613,E2 -15439.613} C_VEL
LIN {X 0,Y 325.726,Z 457.264,A -85,B 0,C 180,E1 -15440.067,E2 -15440.067} C_VEL
LIN {X 0,Y 324.387,Z 447.724,A -85,B 0,C 180,E1 -15441.076,E2 -15441.076} C_VEL
LIN {X 0,Y 321.761,Z 436.02,A -85,B 0,C 180,E1 -15442.114,E2 -15442.114} C_VEL
LIN {X 0,Y 321.128,Z 433.6,A -85,B 0,C 180,E1 -15442.304,E2 -15442.304} C_VEL
LIN {X 0,Y 319.678,Z 430.674,A -85,B 0,C 180,E1 -15442.668,E2 -15442.668} C_VEL
LIN {X 0,Y 317.411,Z 427.46,A -85,B 0,C 180,E1 -15443.443,E2 -15443.443} C_VEL
LIN {X 0,Y 315.381,Z 425.38,A -85,B 0,C 180,E1 -15444.377,E2 -15444.377} C_VEL
LIN {X 0,Y 313.333,Z 423.76,A -85,B 0,C 180,E1 -15445.814,E2 -15445.814} C_VEL
LIN {X 0,Y 312.64,Z 421.954,A -85,B 0,C 180,E1 -15447.303,E2 -15447.303} C_VEL
LIN {X 0,Y 313.199,Z 416.128,A -85,B 0,C 180,E1 -15451.887,E2 -15451.887} C_VEL
LIN {X 0,Y 313.568,Z 412.528,A -85,B 0,C 180,E1 -15454.796,E2 -15454.796} C_VEL
LIN {X 0,Y 313.669,Z 409.227,A -85,B 0,C 180,E1 -15457.611,E2 -15457.611} C_VEL
LIN {X 0,Y 313.386,Z 406.205,A -85,B 0,C 180,E1 -15460.359,E2 -15460.359} C_VEL
LIN {X 0,Y 312.74,Z 402.142,A -85,B 0,C 180,E1 -15464.356,E2 -15464.356} C_VEL
LIN {X 0,Y 312.68,Z 401.541,A -85,B 0,C 180,E1 -15465.11,E2 -15465.11} C_VEL
LIN {X 0,Y 312.682,Z 401.538,A -85,B 0,C 180,E1 -15469.642,E2 -15469.642} C_VEL
LIN {X 0,Y 312.85,Z 401.515,A -85,B 0,C 180,E1 -15472.254,E2 -15472.254} C_VEL
LIN {X 0,Y 312.704,Z 401.536,A -85,B 0,C 180,E1 -15474.843,E2 -15474.843} C_VEL
LIN {X 0,Y 312.94,Z 401.506,A -85,B 0,C 180,E1 -15477.426,E2 -15477.426} C_VEL
LIN {X 0,Y 313.118,Z 401.483,A -85,B 0,C 180,E1 -15480,E2 -15480} C_VEL
LIN {X 0,Y 312.94,Z 401.505,A -85,B 0,C 180,E1 -15482.575,E2 -15482.575} C_VEL
LIN {X 0,Y 312.891,Z 401.505,A -85,B 0,C 180,E1 -15486.449,E2 -15486.449} C_VEL
LIN {X 0,Y 312.766,Z 401.522,A -85,B 0,C 180,E1 -15489.05,E2 -15489.05} C_VEL
LIN {X 0,Y 312.616,Z 401.54,A -85,B 0,C 180,E1 -15492.992,E2 -15492.992} C_VEL
LIN {X 0,Y 312.618,Z 401.539,A -85,B 0,C 180,E1 -15495.651,E2 -15495.651} C_VEL
LIN {X 0,Y 312.591,Z 401.549,A -85,B 0,C 180,E1 -15499.71,E2 -15499.71} C_VEL
LIN {X 0,Y 312.535,Z 401.555,A -85,B 0,C 180,E1 -15502.795,E2 -15502.795} C_VEL
LIN {X 0,Y 312.585,Z 401.549,A -85,B 0,C 180,E1 -15505.938,E2 -15505.938} C_VEL
LIN {X 0,Y 312.527,Z 401.55,A -85,B 0,C 180,E1 -15509.652,E2 -15509.652} C_VEL
LIN {X 0,Y 312.502,Z 401.559,A -85,B 0,C 180,E1 -15513.691,E2 -15513.691} C_VEL
LIN {X 0,Y 312.537,Z 401.556,A -85,B 0,C 180,E1 -15517.384,E2 -15517.384} C_VEL
LIN {X 0,Y 312.513,Z 401.559,A -85,B 0,C 180,E1 -15520.706,E2 -15520.706} C_VEL
LIN {X 0,Y 312.596,Z 401.607,A -85,B 0,C 180,E1 -15523.034,E2 -15523.034} C_VEL
LIN {X 0,Y 313.568,Z 406.413,A -85,B 0,C 180,E1 -15526.754,E2 -15526.754} C_VEL
LIN {X 0,Y 314.615,Z 411.795,A -85,B 0,C 180,E1 -15530.463,E2 -15530.463} C_VEL
LIN {X 0,Y 315.893,Z 418.558,A -85,B 0,C 180,E1 -15534.663,E2 -15534.663} C_VEL
LIN {X 0,Y 316.697,Z 423.543,A -85,B 0,C 180,E1 -15537.489,E2 -15537.489} C_VEL
LIN {X 0,Y 316.243,Z 427.002,A -85,B 0,C 180,E1 -15539.264,E2 -15539.264} C_VEL
LIN {X 0,Y 314.604,Z 435.691,A -85,B 0,C 180,E1 -15543.466,E2 -15543.466} C_VEL
LIN {X 0,Y 313.446,Z 443.033,A -85,B 0,C 180,E1 -15546.891,E2 -15546.891} C_VEL
LIN {X 0,Y 316.353,Z 457.272,A -85,B 0,C 180,E1 -15547.751,E2 -15547.751} C_VEL
LIN {X 0,Y 317.878,Z 469.177,A -85,B 0,C 180,E1 -15548.646,E2 -15548.646} C_VEL
LIN {X 0,Y 318.532,Z 480.405,A -85,B 0,C 180,E1 -15549.669,E2 -15549.669} C_VEL
LIN {X 0,Y 318.336,Z 486.834,A -85,B 0,C 180,E1 -15550.329,E2 -15550.329} C_VEL
LIN {X 0,Y 316.645,Z 498.597,A -85,B 0,C 180,E1 -15551.733,E2 -15551.733} C_VEL
LIN {X 0,Y 315.214,Z 508.035,A -85,B 0,C 180,E1 -15553.155,E2 -15553.155} C_VEL
LIN {X 0,Y 314.06,Z 516.582,A -85,B 0,C 180,E1 -15554.759,E2 -15554.759} C_VEL
LIN {X 0,Y 312.878,Z 524.859,A -85,B 0,C 180,E1 -15556.692,E2 -15556.692} C_VEL
LIN {X 0,Y 311.977,Z 530.478,A -85,B 0,C 180,E1 -15558.306,E2 -15558.306} C_VEL
LIN {X 0,Y 311.101,Z 539.507,A -85,B 0,C 180,E1 -15561.559,E2 -15561.559} C_VEL
LIN {X 0,Y 310.82,Z 543.962,A -85,B 0,C 180,E1 -15563.512,E2 -15563.512} C_VEL
LIN {X 0,Y 310.714,Z 546.295,A -85,B 0,C 180,E1 -15564.812,E2 -15564.812} C_VEL
LIN {X 0,Y 310.733,Z 548.187,A -85,B 0,C 180,E1 -15566.112,E2 -15566.112} C_VEL
LIN {X 0,Y 310.721,Z 549.586,A -85,B 0,C 180,E1 -15567.41,E2 -15567.41} C_VEL
LIN {X 0,Y 310.716,Z 550.559,A -85,B 0,C 180,E1 -15568.707,E2 -15568.707} C_VEL
LIN {X 0,Y 310.725,Z 551.127,A -85,B 0,C 180,E1 -15570.003,E2 -15570.003} C_VEL
LIN {X 0,Y 310.706,Z 551.268,A -85,B 0,C 180,E1 -15571.299,E2 -15571.299} C_VEL
LIN {X 0,Y 310.723,Z 550.964,A -85,B 0,C 180,E1 -15572.596,E2 -15572.596} C_VEL
LIN {X 0,Y 310.732,Z 550.264,A -85,B 0,C 180,E1 -15573.893,E2 -15573.893} C_VEL
LIN {X 0,Y 310.733,Z 548.681,A -85,B 0,C 180,E1 -15575.63,E2 -15575.63} C_VEL
LIN {X 0,Y 311.058,Z 545.64,A -85,B 0,C 180,E1 -15577.794,E2 -15577.794} C_VEL
LIN {X 0,Y 311.566,Z 541.822,A -85,B 0,C 180,E1 -15579.743,E2 -15579.743} C_VEL
LIN {X 0,Y 312.343,Z 536.877,A -85,B 0,C 180,E1 -15581.686,E2 -15581.686} C_VEL
LIN {X 0,Y 313.41,Z 530.673,A -85,B 0,C 180,E1 -15583.621,E2 -15583.621} C_VEL
LIN {X 0,Y 314.884,Z 523.017,A -85,B 0,C 180,E1 -15585.538,E2 -15585.538} C_VEL
LIN {X 0,Y 316.454,Z 513.54,A -85,B 0,C 180,E1 -15587.448,E2 -15587.448} C_VEL
LIN {X 0,Y 318.276,Z 503.832,A -85,B 0,C 180,E1 -15589.011,E2 -15589.011} C_VEL
LIN {X 0,Y 319.946,Z 494.388,A -85,B 0,C 180,E1 -15590.243,E2 -15590.243} C_VEL
LIN {X 0,Y 321.09,Z 485.955,A -85,B 0,C 180,E1 -15591.173,E2 -15591.173} C_VEL
LIN {X 0,Y 321.039,Z 475.37,A -85,B 0,C 180,E1 -15592.261,E2 -15592.261} C_VEL
LIN {X 0,Y 319.893,Z 463.025,A -85,B 0,C 180,E1 -15593.383,E2 -15593.383} C_VEL
LIN {X 0,Y 317.518,Z 449.622,A -85,B 0,C 180,E1 -15594.445,E2 -15594.445} C_VEL
LIN {X 0,Y 313.95,Z 435.86,A -85,B 0,C 180,E1 -15595.436,E2 -15595.436} C_VEL
LIN {X 0,Y 313.903,Z 435.132,A -85,B 0,C 180,E1 -15595.533,E2 -15595.533} C_VEL
LIN {X 0,Y 315.4,Z 426.17,A -85,B 0,C 180,E1 -15599.653,E2 -15599.653} C_VEL
LIN {X 0,Y 316.035,Z 422.22,A -85,B 0,C 180,E1 -15601.509,E2 -15601.509} C_VEL
LIN {X 0,Y 315.903,Z 419.131,A -85,B 0,C 180,E1 -15603.03,E2 -15603.03} C_VEL
LIN {X 0,Y 314.648,Z 412.617,A -85,B 0,C 180,E1 -15606.476,E2 -15606.476} C_VEL
LIN {X 0,Y 313.321,Z 405.736,A -85,B 0,C 180,E1 -15610.302,E2 -15610.302} C_VEL
LIN {X 0,Y 312.524,Z 401.557,A -85,B 0,C 180,E1 -15612.866,E2 -15612.866} C_VEL
LIN {X 0,Y 312.464,Z 401.556,A -85,B 0,C 180,E1 -15616.036,E2 -15616.036} C_VEL
LIN {X 0,Y 312.463,Z 401.559,A -85,B 0,C 180,E1 -15619.886,E2 -15619.886} C_VEL
LIN {X 0,Y 312.542,Z 401.553,A -85,B 0,C 180,E1 -15624.052,E2 -15624.052} C_VEL
LIN {X 0,Y 312.51,Z 401.557,A -85,B 0,C 180,E1 -15627.334,E2 -15627.334} C_VEL
LIN {X 0,Y 312.505,Z 401.56,A -85,B 0,C 180,E1 -15631.295,E2 -15631.295} C_VEL
LIN {X 0,Y 312.524,Z 401.556,A -85,B 0,C 180,E1 -15634.705,E2 -15634.705} C_VEL
LIN {X 0,Y 312.542,Z 401.554,A -85,B 0,C 180,E1 -15638.913,E2 -15638.913} C_VEL
LIN {X 0,Y 312.647,Z 401.542,A -85,B 0,C 180,E1 -15641.656,E2 -15641.656} C_VEL
LIN {X 0,Y 312.702,Z 401.535,A -85,B 0,C 180,E1 -15645.686,E2 -15645.686} C_VEL
LIN {X 0,Y 312.682,Z 401.655,A -85,B 0,C 180,E1 -15647.506,E2 -15647.506} C_VEL
LIN {X 0,Y 313.788,Z 406.31,A -85,B 0,C 180,E1 -15650.979,E2 -15650.979} C_VEL
LIN {X 0,Y 314.487,Z 410.041,A -85,B 0,C 180,E1 -15653.584,E2 -15653.584} C_VEL
LIN {X 0,Y 314.747,Z 413.936,A -85,B 0,C 180,E1 -15656.159,E2 -15656.159} C_VEL
LIN {X 0,Y 314.409,Z 418.072,A -85,B 0,C 180,E1 -15658.719,E2 -15658.719} C_VEL
LIN {X 0,Y 313.511,Z 426.592,A -85,B 0,C 180,E1 -15663.856,E2 -15663.856} C_VEL
LIN {X 0,Y 313.322,Z 429.413,A -85,B 0,C 180,E1 -15665.551,E2 -15665.551} C_VEL
LIN {X 0,Y 317.843,Z 442.52,A -85,B 0,C 180,E1 -15666.785,E2 -15666.785} C_VEL
LIN {X 0,Y 320.901,Z 454.759,A -85,B 0,C 180,E1 -15668.025,E2 -15668.025} C_VEL
LIN {X 0,Y 322.599,Z 465.903,A -85,B 0,C 180,E1 -15669.245,E2 -15669.245} C_VEL
LIN {X 0,Y 322.512,Z 469.957,A -85,B 0,C 180,E1 -15669.683,E2 -15669.683} C_VEL
LIN {X 0,Y 320.836,Z 480.808,A -85,B 0,C 180,E1 -15670.895,E2 -15670.895} C_VEL
LIN {X 0,Y 318.992,Z 491.524,A -85,B 0,C 180,E1 -15672.404,E2 -15672.404} C_VEL
LIN {X 0,Y 317.19,Z 501.291,A -85,B 0,C 180,E1 -15674.106,E2 -15674.106} C_VEL
LIN {X 0,Y 315.506,Z 509.879,A -85,B 0,C 180,E1 -15675.985,E2 -15675.985} C_VEL
LIN {X 0,Y 314.112,Z 516.974,A -85,B 0,C 180,E1 -15677.917,E2 -15677.917} C_VEL
LIN {X 0,Y 313.06,Z 522.18,A -85,B 0,C 180,E1 -15679.678,E2 -15679.678} C_VEL
LIN {X 0,Y 312.054,Z 527.078,A -85,B 0,C 180,E1 -15681.778,E2 -15681.778} C_VEL
LIN {X 0,Y 311.397,Z 530.787,A -85,B 0,C 180,E1 -15683.969,E2 -15683.969} C_VEL
LIN {X 0,Y 311.028,Z 532.566,A -85,B 0,C 180,E1 -15685.424,E2 -15685.424} C_VEL
LIN {X 0,Y 310.734,Z 533.852,A -85,B 0,C 180,E1 -15686.894,E2 -15686.894} C_VEL
LIN {X 0,Y 310.539,Z 534.578,A -85,B 0,C 180,E1 -15688.376,E2 -15688.376} C_VEL
LIN {X 0,Y 310.39,Z 534.701,A -85,B 0,C 180,E1 -15690.634,E2 -15690.634} C_VEL
LIN {X 0,Y 310.408,Z 533.42,A -85,B 0,C 180,E1 -15693.096,E2 -15693.096} C_VEL
LIN {X 0,Y 310.726,Z 530.727,A -85,B 0,C 180,E1 -15695.484,E2 -15695.484} C_VEL
LIN {X 0,Y 311.119,Z 526.8,A -85,B 0,C 180,E1 -15697.753,E2 -15697.753} C_VEL
LIN {X 0,Y 311.594,Z 521.593,A -85,B 0,C 180,E1 -15699.924,E2 -15699.924} C_VEL
LIN {X 0,Y 312.306,Z 514.996,A -85,B 0,C 180,E1 -15702.042,E2 -15702.042} C_VEL
LIN {X 0,Y 313.188,Z 506.87,A -85,B 0,C 180,E1 -15704.101,E2 -15704.101} C_VEL
LIN {X 0,Y 314.295,Z 497.789,A -85,B 0,C 180,E1 -15705.929,E2 -15705.929} C_VEL
LIN {X 0,Y 315.452,Z 487.878,A -85,B 0,C 180,E1 -15707.55,E2 -15707.55} C_VEL
LIN {X 0,Y 316.685,Z 476.889,A -85,B 0,C 180,E1 -15708.985,E2 -15708.985} C_VEL
LIN {X 0,Y 317.816,Z 465.001,A -85,B 0,C 180,E1 -15710.224,E2 -15710.224} C_VEL
LIN {X 0,Y 317.947,Z 461.497,A -85,B 0,C 180,E1 -15710.536,E2 -15710.536} C_VEL
LIN {X 0,Y 316.183,Z 450.289,A -85,B 0,C 180,E1 -15711.508,E2 -15711.508} C_VEL
LIN {X 0,Y 313.758,Z 437.216,A -85,B 0,C 180,E1 -15712.4,E2 -15712.4} C_VEL
LIN {X 0,Y 311.884,Z 427.992,A -85,B 0,C 180,E1 -15712.928,E2 -15712.928} C_VEL
LIN {X 0,Y 312.235,Z 421.95,A -85,B 0,C 180,E1 -15716.389,E2 -15716.389} C_VEL
LIN {X 0,Y 312.563,Z 415.034,A -85,B 0,C 180,E1 -15720.349,E2 -15720.349} C_VEL
LIN {X 0,Y 312.847,Z 408.755,A -85,B 0,C 180,E1 -15723.972,E2 -15723.972} C_VEL
LIN {X 0,Y 313.04,Z 404.963,A -85,B 0,C 180,E1 -15726.162,E2 -15726.162} C_VEL
LIN {X 0,Y 312.666,Z 401.54,A -85,B 0,C 180,E1 -15728.228,E2 -15728.228} C_VEL
LIN {X 0,Y 312.641,Z 401.543,A -85,B 0,C 180,E1 -15731.654,E2 -15731.654} C_VEL
LIN {X 0,Y 312.696,Z 401.535,A -85,B 0,C 180,E1 -15735.684,E2 -15735.684} C_VEL
LIN {X 0,Y 312.699,Z 401.536,A -85,B 0,C 180,E1 -15739.639,E2 -15739.639} C_VEL
LIN {X 0,Y 312.817,Z 401.521,A -85,B 0,C 180,E1 -15742.25,E2 -15742.25} C_VEL
LIN {X 0,Y 312.694,Z 401.54,A -85,B 0,C 180,E1 -15744.839,E2 -15744.839} C_VEL
LIN {X 0,Y 312.686,Z 401.639,A -85,B 0,C 180,E1 -15746.292,E2 -15746.292} C_VEL
LIN {X 0,Y 313.451,Z 404.557,A -85,B 0,C 180,E1 -15748.712,E2 -15748.712} C_VEL
LIN {X 0,Y 313.234,Z 407.888,A -85,B 0,C 180,E1 -15751.283,E2 -15751.283} C_VEL
LIN {X 0,Y 312.608,Z 414.884,A -85,B 0,C 180,E1 -15756.451,E2 -15756.451} C_VEL
LIN {X 0,Y 312.092,Z 420.317,A -85,B 0,C 180,E1 -15760.375,E2 -15760.375} C_VEL
LIN {X 0,Y 311.702,Z 426.019,A -85,B 0,C 180,E1 -15764.397,E2 -15764.397} C_VEL
LIN {X 0,Y 314.333,Z 438.729,A -85,B 0,C 180,E1 -15765.227,E2 -15765.227} C_VEL
LIN {X 0,Y 316.324,Z 450.497,A -85,B 0,C 180,E1 -15766.237,E2 -15766.237} C_VEL
LIN {X 0,Y 316.983,Z 455.504,A -85,B 0,C 180,E1 -15766.749,E2 -15766.749} C_VEL
LIN {X 0,Y 315.902,Z 466.859,A -85,B 0,C 180,E1 -15768.02,E2 -15768.02} C_VEL
LIN {X 0,Y 314.904,Z 476.279,A -85,B 0,C 180,E1 -15769.385,E2 -15769.385} C_VEL
LIN {X 0,Y 313.917,Z 485.06,A -85,B 0,C 180,E1 -15770.987,E2 -15770.987} C_VEL
LIN {X 0,Y 313.034,Z 492.415,A -85,B 0,C 180,E1 -15772.689,E2 -15772.689} C_VEL
LIN {X 0,Y 312.233,Z 498.913,A -85,B 0,C 180,E1 -15774.605,E2 -15774.605} C_VEL
LIN {X 0,Y 311.553,Z 504.506,A -85,B 0,C 180,E1 -15776.814,E2 -15776.814} C_VEL
LIN {X 0,Y 311.144,Z 508.379,A -85,B 0,C 180,E1 -15779.05,E2 -15779.05} C_VEL
LIN {X 0,Y 310.819,Z 510.744,A -85,B 0,C 180,E1 -15781.332,E2 -15781.332} C_VEL
LIN {X 0,Y 310.811,Z 511.547,A -85,B 0,C 180,E1 -15783.214,E2 -15783.214} C_VEL
LIN {X 0,Y 310.869,Z 511.55,A -85,B 0,C 180,E1 -15784.411,E2 -15784.411} C_VEL
LIN {X 0,Y 311.034,Z 510.899,A -85,B 0,C 180,E1 -15785.974,E2 -15785.974} C_VEL
LIN {X 0,Y 311.372,Z 509.246,A -85,B 0,C 180,E1 -15787.816,E2 -15787.816} C_VEL
LIN {X 0,Y 312.013,Z 505.881,A -85,B 0,C 180,E1 -15790.019,E2 -15790.019} C_VEL
LIN {X 0,Y 312.845,Z 501.085,A -85,B 0,C 180,E1 -15792.155,E2 -15792.155} C_VEL
LIN {X 0,Y 313.921,Z 494.646,A -85,B 0,C 180,E1 -15794.242,E2 -15794.242} C_VEL
LIN {X 0,Y 314.97,Z 487.842,A -85,B 0,C 180,E1 -15795.94,E2 -15795.94} C_VEL
LIN {X 0,Y 316.359,Z 479.44,A -85,B 0,C 180,E1 -15797.595,E2 -15797.595} C_VEL
LIN {X 0,Y 317.692,Z 470.293,A -85,B 0,C 180,E1 -15799.012,E2 -15799.012} C_VEL
LIN {X 0,Y 319.048,Z 459.724,A -85,B 0,C 180,E1 -15800.297,E2 -15800.297} C_VEL
LIN {X 0,Y 317.981,Z 450.567,A -85,B 0,C 180,E1 -15801.323,E2 -15801.323} C_VEL
LIN {X 0,Y 315.63,Z 439.282,A -85,B 0,C 180,E1 -15802.412,E2 -15802.412} C_VEL
LIN {X 0,Y 312.3,Z 427.125,A -85,B 0,C 180,E1 -15803.361,E2 -15803.361} C_VEL
LIN {X 0,Y 312.64,Z 421.954,A -85,B 0,C 180,E1 -15807.303,E2 -15807.303} C_VEL
LIN {X 0,Y 312.094,Z 420.714,A -85,B 0,C 180,E1 -15808.357,E2 -15808.357} C_VEL
LIN {X 0,Y 309.43,Z 419.014,A -85,B 0,C 180,E1 -15810.091,E2 -15810.091} C_VEL
LIN {X 0,Y 307.209,Z 417.704,A -85,B 0,C 180,E1 -15811.498,E2 -15811.498} C_VEL
LIN {X 0,Y 306.37,Z 416.553,A -85,B 0,C 180,E1 -15812.579,E2 -15812.579} C_VEL
LIN {X 0,Y 306.365,Z 416.12,A -85,B 0,C 180,E1 -15812.941,E2 -15812.941} C_VEL
LIN {X 0,Y 306.624,Z 412.934,A -85,B 0,C 180,E1 -15815.634,E2 -15815.634} C_VEL
LIN {X 0,Y 306.628,Z 409.727,A -85,B 0,C 180,E1 -15818.487,E2 -15818.487} C_VEL
LIN {X 0,Y 306.314,Z 406.843,A -85,B 0,C 180,E1 -15821.264,E2 -15821.264} C_VEL
LIN {X 0,Y 305.654,Z 402.516,A -85,B 0,C 180,E1 -15825.69,E2 -15825.69} C_VEL
LIN {X 0,Y 305.619,Z 402.419,A -85,B 0,C 180,E1 -15829.4,E2 -15829.4} C_VEL
LIN {X 0,Y 305.791,Z 402.394,A -85,B 0,C 180,E1 -15832.074,E2 -15832.074} C_VEL
LIN {X 0,Y 305.675,Z 402.411,A -85,B 0,C 180,E1 -15834.724,E2 -15834.724} C_VEL
LIN {X 0,Y 305.942,Z 402.372,A -85,B 0,C 180,E1 -15838.684,E2 -15838.684} C_VEL
LIN {X 0,Y 306.07,Z 402.361,A -85,B 0,C 180,E1 -15840,E2 -15840} C_VEL
LIN {X 0,Y 305.887,Z 402.384,A -85,B 0,C 180,E1 -15842.634,E2 -15842.634} C_VEL
LIN {X 0,Y 305.833,Z 402.383,A -85,B 0,C 180,E1 -15846.598,E2 -15846.598} C_VEL
LIN {X 0,Y 305.715,Z 402.399,A -85,B 0,C 180,E1 -15849.261,E2 -15849.261} C_VEL
LIN {X 0,Y 305.57,Z 402.419,A -85,B 0,C 180,E1 -15853.297,E2 -15853.297} C_VEL
LIN {X 0,Y 305.574,Z 402.417,A -85,B 0,C 180,E1 -15856.022,E2 -15856.022} C_VEL
LIN {X 0,Y 305.584,Z 402.419,A -85,B 0,C 180,E1 -15859.461,E2 -15859.461} C_VEL
LIN {X 0,Y 305.505,Z 402.432,A -85,B 0,C 180,E1 -15863.058,E2 -15863.058} C_VEL
LIN {X 0,Y 305.53,Z 402.425,A -85,B 0,C 180,E1 -15866.23,E2 -15866.23} C_VEL
LIN {X 0,Y 305.478,Z 402.431,A -85,B 0,C 180,E1 -15869.052,E2 -15869.052} C_VEL
LIN {X 0,Y 305.448,Z 402.438,A -85,B 0,C 180,E1 -15873.519,E2 -15873.519} C_VEL
LIN {X 0,Y 305.486,Z 402.433,A -85,B 0,C 180,E1 -15876.738,E2 -15876.738} C_VEL
LIN {X 0,Y 305.472,Z 402.436,A -85,B 0,C 180,E1 -15880.61,E2 -15880.61} C_VEL
LIN {X 0,Y 305.524,Z 402.51,A -85,B 0,C 180,E1 -15882.044,E2 -15882.044} C_VEL
LIN {X 0,Y 306.393,Z 406.495,A -85,B 0,C 180,E1 -15885.323,E2 -15885.323} C_VEL
LIN {X 0,Y 307.352,Z 411.468,A -85,B 0,C 180,E1 -15888.99,E2 -15888.99} C_VEL
LIN {X 0,Y 308.446,Z 417.349,A -85,B 0,C 180,E1 -15892.891,E2 -15892.891} C_VEL
LIN {X 0,Y 309.477,Z 422.772,A -85,B 0,C 180,E1 -15896.199,E2 -15896.199} C_VEL
LIN {X 0,Y 309.764,Z 425.677,A -85,B 0,C 180,E1 -15897.832,E2 -15897.832} C_VEL
LIN {X 0,Y 308.317,Z 432.719,A -85,B 0,C 180,E1 -15901.404,E2 -15901.404} C_VEL
LIN {X 0,Y 306.794,Z 441.431,A -85,B 0,C 180,E1 -15905.652,E2 -15905.652} C_VEL
LIN {X 0,Y 306.564,Z 442.816,A -85,B 0,C 180,E1 -15906.306,E2 -15906.306} C_VEL
LIN {X 0,Y 309.443,Z 456.32,A -85,B 0,C 180,E1 -15907.138,E2 -15907.138} C_VEL
LIN {X 0,Y 311.087,Z 468.461,A -85,B 0,C 180,E1 -15908.075,E2 -15908.075} C_VEL
LIN {X 0,Y 311.823,Z 480.578,A -85,B 0,C 180,E1 -15909.211,E2 -15909.211} C_VEL
LIN {X 0,Y 311.465,Z 488.319,A -85,B 0,C 180,E1 -15910.048,E2 -15910.048} C_VEL
LIN {X 0,Y 309.914,Z 498.562,A -85,B 0,C 180,E1 -15911.321,E2 -15911.321} C_VEL
LIN {X 0,Y 308.4,Z 507.924,A -85,B 0,C 180,E1 -15912.771,E2 -15912.771} C_VEL
LIN {X 0,Y 307.2,Z 516.395,A -85,B 0,C 180,E1 -15914.41,E2 -15914.41} C_VEL
LIN {X 0,Y 305.94,Z 524.64,A -85,B 0,C 180,E1 -15916.385,E2 -15916.385} C_VEL
LIN {X 0,Y 304.996,Z 530.228,A -85,B 0,C 180,E1 -15918.034,E2 -15918.034} C_VEL
LIN {X 0,Y 304.333,Z 535.678,A -85,B 0,C 180,E1 -15920.029,E2 -15920.029} C_VEL
LIN {X 0,Y 303.824,Z 542.148,A -85,B 0,C 180,E1 -15922.694,E2 -15922.694} C_VEL
LIN {X 0,Y 303.638,Z 545.91,A -85,B 0,C 180,E1 -15924.691,E2 -15924.691} C_VEL
LIN {X 0,Y 303.644,Z 547.831,A -85,B 0,C 180,E1 -15926.021,E2 -15926.021} C_VEL
LIN {X 0,Y 303.644,Z 549.288,A -85,B 0,C 180,E1 -15927.35,E2 -15927.35} C_VEL
LIN {X 0,Y 303.629,Z 550.288,A -85,B 0,C 180,E1 -15928.677,E2 -15928.677} C_VEL
LIN {X 0,Y 303.637,Z 550.885,A -85,B 0,C 180,E1 -15930.003,E2 -15930.003} C_VEL
LIN {X 0,Y 303.62,Z 551.076,A -85,B 0,C 180,E1 -15931.329,E2 -15931.329} C_VEL
LIN {X 0,Y 303.645,Z 550.816,A -85,B 0,C 180,E1 -15932.656,E2 -15932.656} C_VEL
LIN {X 0,Y 303.644,Z 550.148,A -85,B 0,C 180,E1 -15933.984,E2 -15933.984} C_VEL
LIN {X 0,Y 303.644,Z 548.835,A -85,B 0,C 180,E1 -15935.577,E2 -15935.577} C_VEL
LIN {X 0,Y 304.013,Z 545.649,A -85,B 0,C 180,E1 -15937.976,E2 -15937.976} C_VEL
LIN {X 0,Y 304.538,Z 541.897,A -85,B 0,C 180,E1 -15939.97,E2 -15939.97} C_VEL
LIN {X 0,Y 305.352,Z 537.043,A -85,B 0,C 180,E1 -15941.958,E2 -15941.958} C_VEL
LIN {X 0,Y 306.53,Z 530.957,A -85,B 0,C 180,E1 -15943.933,E2 -15943.933} C_VEL
LIN {X 0,Y 308.062,Z 523.443,A -85,B 0,C 180,E1 -15945.891,E2 -15945.891} C_VEL
LIN {X 0,Y 309.72,Z 514.114,A -85,B 0,C 180,E1 -15947.84,E2 -15947.84} C_VEL
LIN {X 0,Y 311.753,Z 503.522,A -85,B 0,C 180,E1 -15949.595,E2 -15949.595} C_VEL
LIN {X 0,Y 313.825,Z 492.752,A -85,B 0,C 180,E1 -15950.999,E2 -15950.999} C_VEL
LIN {X 0,Y 314.667,Z 485.753,A -85,B 0,C 180,E1 -15951.799,E2 -15951.799} C_VEL
LIN {X 0,Y 314.621,Z 476.218,A -85,B 0,C 180,E1 -15952.825,E2 -15952.825} C_VEL
LIN {X 0,Y 313.686,Z 464.836,A -85,B 0,C 180,E1 -15953.918,E2 -15953.918} C_VEL
LIN {X 0,Y 311.377,Z 451.198,A -85,B 0,C 180,E1 -15955.075,E2 -15955.075} C_VEL
LIN {X 0,Y 307.85,Z 437.6,A -85,B 0,C 180,E1 -15956.138,E2 -15956.138} C_VEL
LIN {X 0,Y 307.242,Z 435.174,A -85,B 0,C 180,E1 -15956.345,E2 -15956.345} C_VEL
LIN {X 0,Y 307.256,Z 433.444,A -85,B 0,C 180,E1 -15956.742,E2 -15956.742} C_VEL
LIN {X 0,Y 308.794,Z 424.876,A -85,B 0,C 180,E1 -15960.806,E2 -15960.806} C_VEL
LIN {X 0,Y 308.986,Z 421.073,A -85,B 0,C 180,E1 -15962.692,E2 -15962.692} C_VEL
LIN {X 0,Y 308.033,Z 415.657,A -85,B 0,C 180,E1 -15965.579,E2 -15965.579} C_VEL
LIN {X 0,Y 306.916,Z 409.766,A -85,B 0,C 180,E1 -15968.871,E2 -15968.871} C_VEL
LIN {X 0,Y 305.462,Z 402.453,A -85,B 0,C 180,E1 -15973.227,E2 -15973.227} C_VEL
LIN {X 0,Y 305.443,Z 402.438,A -85,B 0,C 180,E1 -15977.419,E2 -15977.419} C_VEL
LIN {X 0,Y 305.468,Z 402.427,A -85,B 0,C 180,E1 -15981.596,E2 -15981.596} C_VEL
LIN {X 0,Y 305.47,Z 402.435,A -85,B 0,C 180,E1 -15984.887,E2 -15984.887} C_VEL
LIN {X 0,Y 305.45,Z 402.437,A -85,B 0,C 180,E1 -15988.359,E2 -15988.359} C_VEL
LIN {X 0,Y 305.471,Z 402.436,A -85,B 0,C 180,E1 -15991.108,E2 -15991.108} C_VEL
LIN {X 0,Y 305.486,Z 402.433,A -85,B 0,C 180,E1 -15994.08,E2 -15994.08} C_VEL
LIN {X 0,Y 305.478,Z 402.435,A -85,B 0,C 180,E1 -15998.401,E2 -15998.401} C_VEL
LIN {X 0,Y 305.588,Z 402.421,A -85,B 0,C 180,E1 -16001.217,E2 -16001.217} C_VEL
LIN {X 0,Y 305.658,Z 402.415,A -85,B 0,C 180,E1 -16005.349,E2 -16005.349} C_VEL
LIN {X 0,Y 305.658,Z 402.62,A -85,B 0,C 180,E1 -16006.368,E2 -16006.368} C_VEL
LIN {X 0,Y 306.758,Z 407.36,A -85,B 0,C 180,E1 -16010.124,E2 -16010.124} C_VEL
LIN {X 0,Y 307.669,Z 411.876,A -85,B 0,C 180,E1 -16013.441,E2 -16013.441} C_VEL
LIN {X 0,Y 307.922,Z 415.8,A -85,B 0,C 180,E1 -16016.073,E2 -16016.073} C_VEL
LIN {X 0,Y 307.544,Z 419.92,A -85,B 0,C 180,E1 -16018.69,E2 -16018.69} C_VEL
LIN {X 0,Y 306.582,Z 428.421,A -85,B 0,C 180,E1 -16023.943,E2 -16023.943} C_VEL
LIN {X 0,Y 306.51,Z 429.705,A -85,B 0,C 180,E1 -16024.685,E2 -16024.685} C_VEL
LIN {X 0,Y 311.347,Z 443.316,A -85,B 0,C 180,E1 -16026.066,E2 -16026.066} C_VEL
LIN {X 0,Y 314.254,Z 454.664,A -85,B 0,C 180,E1 -16027.281,E2 -16027.281} C_VEL
LIN {X 0,Y 316.119,Z 466.369,A -85,B 0,C 180,E1 -16028.63,E2 -16028.63} C_VEL
LIN {X 0,Y 316.186,Z 470.627,A -85,B 0,C 180,E1 -16029.121,E2 -16029.121} C_VEL
LIN {X 0,Y 314.387,Z 481.588,A -85,B 0,C 180,E1 -16030.382,E2 -16030.382} C_VEL
LIN {X 0,Y 312.336,Z 492.814,A -85,B 0,C 180,E1 -16032.013,E2 -16032.013} C_VEL
LIN {X 0,Y 310.314,Z 502.899,A -85,B 0,C 180,E1 -16033.87,E2 -16033.87} C_VEL
LIN {X 0,Y 308.537,Z 511.5,A -85,B 0,C 180,E1 -16035.863,E2 -16035.863} C_VEL
LIN {X 0,Y 306.936,Z 518.818,A -85,B 0,C 180,E1 -16038.005,E2 -16038.005} C_VEL
LIN {X 0,Y 305.72,Z 524.579,A -85,B 0,C 180,E1 -16040.171,E2 -16040.171} C_VEL
LIN {X 0,Y 305.024,Z 527.681,A -85,B 0,C 180,E1 -16041.632,E2 -16041.632} C_VEL
LIN {X 0,Y 304.546,Z 530.166,A -85,B 0,C 180,E1 -16043.098,E2 -16043.098} C_VEL
LIN {X 0,Y 303.909,Z 533.208,A -85,B 0,C 180,E1 -16045.589,E2 -16045.589} C_VEL
LIN {X 0,Y 303.446,Z 534.83,A -85,B 0,C 180,E1 -16048.342,E2 -16048.342} C_VEL
LIN {X 0,Y 303.308,Z 534.77,A -85,B 0,C 180,E1 -16050.978,E2 -16050.978} C_VEL
LIN {X 0,Y 303.34,Z 533.214,A -85,B 0,C 180,E1 -16053.477,E2 -16053.477} C_VEL
LIN {X 0,Y 303.691,Z 530.297,A -85,B 0,C 180,E1 -16055.904,E2 -16055.904} C_VEL
LIN {X 0,Y 304.106,Z 526.086,A -85,B 0,C 180,E1 -16058.207,E2 -16058.207} C_VEL
LIN {X 0,Y 304.61,Z 520.654,A -85,B 0,C 180,E1 -16060.411,E2 -16060.411} C_VEL
LIN {X 0,Y 305.428,Z 513.751,A -85,B 0,C 180,E1 -16062.577,E2 -16062.577} C_VEL
LIN {X 0,Y 306.38,Z 505.258,A -85,B 0,C 180,E1 -16064.672,E2 -16064.672} C_VEL
LIN {X 0,Y 307.501,Z 496.417,A -85,B 0,C 180,E1 -16066.428,E2 -16066.428} C_VEL
LIN {X 0,Y 308.636,Z 486.788,A -85,B 0,C 180,E1 -16067.979,E2 -16067.979} C_VEL
LIN {X 0,Y 309.962,Z 475.314,A -85,B 0,C 180,E1 -16069.471,E2 -16069.471} C_VEL
LIN {X 0,Y 311.02,Z 464.178,A -85,B 0,C 180,E1 -16070.62,E2 -16070.62} C_VEL
LIN {X 0,Y 310.035,Z 455.633,A -85,B 0,C 180,E1 -16071.418,E2 -16071.418} C_VEL
LIN {X 0,Y 307.716,Z 442.482,A -85,B 0,C 180,E1 -16072.442,E2 -16072.442} C_VEL
LIN {X 0,Y 304.991,Z 429.108,A -85,B 0,C 180,E1 -16073.234,E2 -16073.234} C_VEL
LIN {X 0,Y 304.877,Z 428.152,A -85,B 0,C 180,E1 -16073.307,E2 -16073.307} C_VEL
LIN {X 0,Y 305.231,Z 421.367,A -85,B 0,C 180,E1 -16077.239,E2 -16077.239} C_VEL
LIN {X 0,Y 305.564,Z 414.707,A -85,B 0,C 180,E1 -16081.116,E2 -16081.116} C_VEL
LIN {X 0,Y 306.015,Z 407.084,A -85,B 0,C 180,E1 -16085.579,E2 -16085.579} C_VEL
LIN {X 0,Y 305.712,Z 402.945,A -85,B 0,C 180,E1 -16088.061,E2 -16088.061} C_VEL
LIN {X 0,Y 305.621,Z 402.418,A -85,B 0,C 180,E1 -16088.409,E2 -16088.409} C_VEL
LIN {X 0,Y 305.594,Z 402.42,A -85,B 0,C 180,E1 -16091.215,E2 -16091.215} C_VEL
LIN {X 0,Y 305.651,Z 402.414,A -85,B 0,C 180,E1 -16095.346,E2 -16095.346} C_VEL
LIN {X 0,Y 305.636,Z 402.416,A -85,B 0,C 180,E1 -16099.397,E2 -16099.397} C_VEL
LIN {X 0,Y 305.764,Z 402.399,A -85,B 0,C 180,E1 -16102.07,E2 -16102.07} C_VEL
LIN {X 0,Y 305.664,Z 402.415,A -85,B 0,C 180,E1 -16104.72,E2 -16104.72} C_VEL
LIN {X 0,Y 305.648,Z 402.535,A -85,B 0,C 180,E1 -16106.042,E2 -16106.042} C_VEL
LIN {X 0,Y 306.455,Z 405.677,A -85,B 0,C 180,E1 -16108.683,E2 -16108.683} C_VEL
LIN {X 0,Y 306.203,Z 409.04,A -85,B 0,C 180,E1 -16111.312,E2 -16111.312} C_VEL
LIN {X 0,Y 305.546,Z 416.039,A -85,B 0,C 180,E1 -16116.601,E2 -16116.601} C_VEL
LIN {X 0,Y 305.012,Z 421.537,A -85,B 0,C 180,E1 -16120.619,E2 -16120.619} C_VEL
LIN {X 0,Y 304.675,Z 426.22,A -85,B 0,C 180,E1 -16123.996,E2 -16123.996} C_VEL
LIN {X 0,Y 307.255,Z 438.462,A -85,B 0,C 180,E1 -16124.802,E2 -16124.802} C_VEL
LIN {X 0,Y 309.209,Z 450.205,A -85,B 0,C 180,E1 -16125.824,E2 -16125.824} C_VEL
LIN {X 0,Y 310.065,Z 456.774,A -85,B 0,C 180,E1 -16126.517,E2 -16126.517} C_VEL
LIN {X 0,Y 308.985,Z 467.484,A -85,B 0,C 180,E1 -16127.756,E2 -16127.756} C_VEL
LIN {X 0,Y 307.838,Z 477.901,A -85,B 0,C 180,E1 -16129.328,E2 -16129.328} C_VEL
LIN {X 0,Y 306.905,Z 485.832,A -85,B 0,C 180,E1 -16130.845,E2 -16130.845} C_VEL
LIN {X 0,Y 305.972,Z 493.268,A -85,B 0,C 180,E1 -16132.624,E2 -16132.624} C_VEL
LIN {X 0,Y 305.195,Z 499.364,A -85,B 0,C 180,E1 -16134.484,E2 -16134.484} C_VEL
LIN {X 0,Y 304.489,Z 504.945,A -85,B 0,C 180,E1 -16136.745,E2 -16136.745} C_VEL
LIN {X 0,Y 304.052,Z 508.812,A -85,B 0,C 180,E1 -16139.035,E2 -16139.035} C_VEL
LIN {X 0,Y 303.751,Z 511,A -85,B 0,C 180,E1 -16141.121,E2 -16141.121} C_VEL
LIN {X 0,Y 303.743,Z 512.01,A -85,B 0,C 180,E1 -16143.596,E2 -16143.596} C_VEL
LIN {X 0,Y 303.967,Z 511.381,A -85,B 0,C 180,E1 -16145.98,E2 -16145.98} C_VEL
LIN {X 0,Y 304.405,Z 509.313,A -85,B 0,C 180,E1 -16148.282,E2 -16148.282} C_VEL
LIN {X 0,Y 305.113,Z 505.787,A -85,B 0,C 180,E1 -16150.525,E2 -16150.525} C_VEL
LIN {X 0,Y 305.994,Z 500.81,A -85,B 0,C 180,E1 -16152.696,E2 -16152.696} C_VEL
LIN {X 0,Y 307.009,Z 495.353,A -85,B 0,C 180,E1 -16154.488,E2 -16154.488} C_VEL
LIN {X 0,Y 308.204,Z 487.969,A -85,B 0,C 180,E1 -16156.38,E2 -16156.38} C_VEL
LIN {X 0,Y 309.645,Z 479.802,A -85,B 0,C 180,E1 -16158.015,E2 -16158.015} C_VEL
LIN {X 0,Y 311.039,Z 470.675,A -85,B 0,C 180,E1 -16159.457,E2 -16159.457} C_VEL
LIN {X 0,Y 312.383,Z 460.352,A -85,B 0,C 180,E1 -16160.747,E2 -16160.747} C_VEL
LIN {X 0,Y 310.951,Z 449.632,A -85,B 0,C 180,E1 -16161.984,E2 -16161.984} C_VEL
LIN {X 0,Y 308.316,Z 437.681,A -85,B 0,C 180,E1 -16163.145,E2 -16163.145} C_VEL
LIN {X 0,Y 305.337,Z 427.372,A -85,B 0,C 180,E1 -16163.995,E2 -16163.995} C_VEL
LIN {X 0,Y 305.649,Z 423.04,A -85,B 0,C 180,E1 -16167.357,E2 -16167.357} C_VEL
LIN {X 0,Y 306.076,Z 418.309,A -85,B 0,C 180,E1 -16171.172,E2 -16171.172} C_VEL
LIN {X 0,Y 306.365,Z 416.12,A -85,B 0,C 180,E1 -16172.941,E2 -16172.941} C_VEL
LIN {X 0,Y 306.19,Z 415.311,A -85,B 0,C 180,E1 -16173.66,E2 -16173.66} C_VEL
LIN {X 0,Y 304.992,Z 414.303,A -85,B 0,C 180,E1 -16174.731,E2 -16174.731} C_VEL
LIN {X 0,Y 300.792,Z 412.339,A -85,B 0,C 180,E1 -16177.234,E2 -16177.234} C_VEL
LIN {X 0,Y 299.723,Z 411.362,A -85,B 0,C 180,E1 -16178.344,E2 -16178.344} C_VEL
LIN {X 0,Y 299.623,Z 410.985,A -85,B 0,C 180,E1 -16178.719,E2 -16178.719} C_VEL
LIN {X 0,Y 299.213,Z 407.433,A -85,B 0,C 180,E1 -16182.221,E2 -16182.221} C_VEL
LIN {X 0,Y 298.845,Z 404.818,A -85,B 0,C 180,E1 -16185.008,E2 -16185.008} C_VEL
LIN {X 0,Y 298.541,Z 403.299,A -85,B 0,C 180,E1 -16186.731,E2 -16186.731} C_VEL
LIN {X 0,Y 298.726,Z 403.279,A -85,B 0,C 180,E1 -16191.129,E2 -16191.129} C_VEL
LIN {X 0,Y 298.777,Z 403.271,A -85,B 0,C 180,E1 -16193.246,E2 -16193.246} C_VEL
LIN {X 0,Y 298.836,Z 403.263,A -85,B 0,C 180,E1 -16197.305,E2 -16197.305} C_VEL
LIN {X 0,Y 299.022,Z 403.239,A -85,B 0,C 180,E1 -16200,E2 -16200} C_VEL
LIN {X 0,Y 298.835,Z 403.262,A -85,B 0,C 180,E1 -16202.696,E2 -16202.696} C_VEL
LIN {X 0,Y 298.778,Z 403.262,A -85,B 0,C 180,E1 -16206.755,E2 -16206.755} C_VEL
LIN {X 0,Y 298.66,Z 403.277,A -85,B 0,C 180,E1 -16209.482,E2 -16209.482} C_VEL
LIN {X 0,Y 298.533,Z 403.298,A -85,B 0,C 180,E1 -16213.617,E2 -16213.617} C_VEL
LIN {X 0,Y 298.529,Z 403.297,A -85,B 0,C 180,E1 -16216.41,E2 -16216.41} C_VEL
LIN {X 0,Y 298.514,Z 403.301,A -85,B 0,C 180,E1 -16219.668,E2 -16219.668} C_VEL
LIN {X 0,Y 298.453,Z 403.306,A -85,B 0,C 180,E1 -16223.599,E2 -16223.599} C_VEL
LIN {X 0,Y 298.471,Z 403.302,A -85,B 0,C 180,E1 -16226.577,E2 -16226.577} C_VEL
LIN {X 0,Y 298.403,Z 403.309,A -85,B 0,C 180,E1 -16229.643,E2 -16229.643} C_VEL
LIN {X 0,Y 298.379,Z 403.313,A -85,B 0,C 180,E1 -16232.803,E2 -16232.803} C_VEL
LIN {X 0,Y 298.454,Z 403.309,A -85,B 0,C 180,E1 -16236.816,E2 -16236.816} C_VEL
LIN {X 0,Y 298.431,Z 403.422,A -85,B 0,C 180,E1 -16240.989,E2 -16240.989} C_VEL
LIN {X 0,Y 299.408,Z 407.741,A -85,B 0,C 180,E1 -16244.765,E2 -16244.765} C_VEL
LIN {X 0,Y 300.367,Z 412.583,A -85,B 0,C 180,E1 -16248.482,E2 -16248.482} C_VEL
LIN {X 0,Y 301.247,Z 417.377,A -85,B 0,C 180,E1 -16251.779,E2 -16251.779} C_VEL
LIN {X 0,Y 302.316,Z 422.909,A -85,B 0,C 180,E1 -16255.33,E2 -16255.33} C_VEL
LIN {X 0,Y 302.808,Z 427.012,A -85,B 0,C 180,E1 -16257.741,E2 -16257.741} C_VEL
LIN {X 0,Y 301.276,Z 434.131,A -85,B 0,C 180,E1 -16261.435,E2 -16261.435} C_VEL
LIN {X 0,Y 299.75,Z 442.55,A -85,B 0,C 180,E1 -16265.652,E2 -16265.652} C_VEL
LIN {X 0,Y 302.728,Z 456.563,A -85,B 0,C 180,E1 -16266.574,E2 -16266.574} C_VEL
LIN {X 0,Y 304.412,Z 469.142,A -85,B 0,C 180,E1 -16267.598,E2 -16267.598} C_VEL
LIN {X 0,Y 305.126,Z 480.751,A -85,B 0,C 180,E1 -16268.733,E2 -16268.733} C_VEL
LIN {X 0,Y 304.814,Z 488.392,A -85,B 0,C 180,E1 -16269.594,E2 -16269.594} C_VEL
LIN {X 0,Y 303.185,Z 498.562,A -85,B 0,C 180,E1 -16270.891,E2 -16270.891} C_VEL
LIN {X 0,Y 301.609,Z 507.852,A -85,B 0,C 180,E1 -16272.37,E2 -16272.37} C_VEL
LIN {X 0,Y 300.348,Z 516.262,A -85,B 0,C 180,E1 -16274.045,E2 -16274.045} C_VEL
LIN {X 0,Y 299.021,Z 524.449,A -85,B 0,C 180,E1 -16276.063,E2 -16276.063} C_VEL
LIN {X 0,Y 298.017,Z 529.992,A -85,B 0,C 180,E1 -16277.75,E2 -16277.75} C_VEL
LIN {X 0,Y 297.32,Z 535.393,A -85,B 0,C 180,E1 -16279.792,E2 -16279.792} C_VEL
LIN {X 0,Y 296.682,Z 543.082,A -85,B 0,C 180,E1 -16283.201,E2 -16283.201} C_VEL
LIN {X 0,Y 296.552,Z 545.489,A -85,B 0,C 180,E1 -16284.564,E2 -16284.564} C_VEL
LIN {X 0,Y 296.559,Z 547.448,A -85,B 0,C 180,E1 -16285.926,E2 -16285.926} C_VEL
LIN {X 0,Y 296.567,Z 548.969,A -85,B 0,C 180,E1 -16287.286,E2 -16287.286} C_VEL
LIN {X 0,Y 296.546,Z 550.009,A -85,B 0,C 180,E1 -16288.645,E2 -16288.645} C_VEL
LIN {X 0,Y 296.55,Z 550.639,A -85,B 0,C 180,E1 -16290.003,E2 -16290.003} C_VEL
LIN {X 0,Y 296.538,Z 550.867,A -85,B 0,C 180,E1 -16291.361,E2 -16291.361} C_VEL
LIN {X 0,Y 296.568,Z 550.668,A -85,B 0,C 180,E1 -16292.72,E2 -16292.72} C_VEL
LIN {X 0,Y 296.54,Z 550.03,A -85,B 0,C 180,E1 -16294.08,E2 -16294.08} C_VEL
LIN {X 0,Y 296.696,Z 547.564,A -85,B 0,C 180,E1 -16296.805,E2 -16296.805} C_VEL
LIN {X 0,Y 297.127,Z 544.58,A -85,B 0,C 180,E1 -16298.847,E2 -16298.847} C_VEL
LIN {X 0,Y 297.777,Z 540.568,A -85,B 0,C 180,E1 -16300.886,E2 -16300.886} C_VEL
LIN {X 0,Y 298.937,Z 534.42,A -85,B 0,C 180,E1 -16303.254,E2 -16303.254} C_VEL
LIN {X 0,Y 300.437,Z 527.737,A -85,B 0,C 180,E1 -16305.261,E2 -16305.261} C_VEL
LIN {X 0,Y 302.023,Z 519.73,A -85,B 0,C 180,E1 -16307.217,E2 -16307.217} C_VEL
LIN {X 0,Y 303.732,Z 511.243,A -85,B 0,C 180,E1 -16308.904,E2 -16308.904} C_VEL
LIN {X 0,Y 305.785,Z 501.124,A -85,B 0,C 180,E1 -16310.52,E2 -16310.52} C_VEL
LIN {X 0,Y 307.944,Z 489.942,A -85,B 0,C 180,E1 -16311.948,E2 -16311.948} C_VEL
LIN {X 0,Y 308.402,Z 480.32,A -85,B 0,C 180,E1 -16313.054,E2 -16313.054} C_VEL
LIN {X 0,Y 307.557,Z 467.114,A -85,B 0,C 180,E1 -16314.426,E2 -16314.426} C_VEL
LIN {X 0,Y 305.586,Z 453.934,A -85,B 0,C 180,E1 -16315.639,E2 -16315.639} C_VEL
LIN {X 0,Y 302.143,Z 440.073,A -85,B 0,C 180,E1 -16316.795,E2 -16316.795} C_VEL
LIN {X 0,Y 300.749,Z 435.107,A -85,B 0,C 180,E1 -16317.251,E2 -16317.251} C_VEL
LIN {X 0,Y 300.713,Z 431.472,A -85,B 0,C 180,E1 -16318.154,E2 -16318.154} C_VEL
LIN {X 0,Y 301.979,Z 424.492,A -85,B 0,C 180,E1 -16321.58,E2 -16321.58} C_VEL
LIN {X 0,Y 301.925,Z 421.604,A -85,B 0,C 180,E1 -16323.071,E2 -16323.071} C_VEL
LIN {X 0,Y 300.749,Z 415.381,A -85,B 0,C 180,E1 -16326.507,E2 -16326.507} C_VEL
LIN {X 0,Y 299.512,Z 409.035,A -85,B 0,C 180,E1 -16330.189,E2 -16330.189} C_VEL
LIN {X 0,Y 298.4,Z 403.316,A -85,B 0,C 180,E1 -16333.839,E2 -16333.839} C_VEL
LIN {X 0,Y 298.378,Z 403.313,A -85,B 0,C 180,E1 -16336.916,E2 -16336.916} C_VEL
LIN {X 0,Y 298.393,Z 403.312,A -85,B 0,C 180,E1 -16341.012,E2 -16341.012} C_VEL
LIN {X 0,Y 298.413,Z 403.313,A -85,B 0,C 180,E1 -16343.929,E2 -16343.929} C_VEL
LIN {X 0,Y 298.401,Z 403.314,A -85,B 0,C 180,E1 -16347.2,E2 -16347.2} C_VEL
LIN {X 0,Y 298.378,Z 403.318,A -85,B 0,C 180,E1 -16350.637,E2 -16350.637} C_VEL
LIN {X 0,Y 298.421,Z 403.312,A -85,B 0,C 180,E1 -16354.918,E2 -16354.918} C_VEL
LIN {X 0,Y 298.441,Z 403.312,A -85,B 0,C 180,E1 -16359.314,E2 -16359.314} C_VEL
LIN {X 0,Y 298.543,Z 403.3,A -85,B 0,C 180,E1 -16362.179,E2 -16362.179} C_VEL
LIN {X 0,Y 298.594,Z 403.318,A -85,B 0,C 180,E1 -16364.806,E2 -16364.806} C_VEL
LIN {X 0,Y 299.358,Z 406.796,A -85,B 0,C 180,E1 -16367.801,E2 -16367.801} C_VEL
LIN {X 0,Y 300.173,Z 410.222,A -85,B 0,C 180,E1 -16370.567,E2 -16370.567} C_VEL
LIN {X 0,Y 300.889,Z 413.847,A -85,B 0,C 180,E1 -16373.293,E2 -16373.293} C_VEL
LIN {X 0,Y 301.112,Z 417.668,A -85,B 0,C 180,E1 -16375.984,E2 -16375.984} C_VEL
LIN {X 0,Y 300.676,Z 421.796,A -85,B 0,C 180,E1 -16378.66,E2 -16378.66} C_VEL
LIN {X 0,Y 299.694,Z 429.828,A -85,B 0,C 180,E1 -16383.739,E2 -16383.739} C_VEL
LIN {X 0,Y 300.993,Z 433.32,A -85,B 0,C 180,E1 -16384.1,E2 -16384.1} C_VEL
LIN {X 0,Y 304.946,Z 444.356,A -85,B 0,C 180,E1 -16385.325,E2 -16385.325} C_VEL
LIN {X 0,Y 308.013,Z 456.415,A -85,B 0,C 180,E1 -16386.697,E2 -16386.697} C_VEL
LIN {X 0,Y 309.685,Z 467.038,A -85,B 0,C 180,E1 -16387.99,E2 -16387.99} C_VEL
LIN {X 0,Y 309.956,Z 470.862,A -85,B 0,C 180,E1 -16388.475,E2 -16388.475} C_VEL
LIN {X 0,Y 308.025,Z 482.075,A -85,B 0,C 180,E1 -16389.803,E2 -16389.803} C_VEL
LIN {X 0,Y 305.935,Z 492.997,A -85,B 0,C 180,E1 -16391.427,E2 -16391.427} C_VEL
LIN {X 0,Y 304.114,Z 501.683,A -85,B 0,C 180,E1 -16393.021,E2 -16393.021} C_VEL
LIN {X 0,Y 302.319,Z 509.633,A -85,B 0,C 180,E1 -16394.816,E2 -16394.816} C_VEL
LIN {X 0,Y 300.797,Z 516.312,A -85,B 0,C 180,E1 -16396.669,E2 -16396.669} C_VEL
LIN {X 0,Y 299.58,Z 521.59,A -85,B 0,C 180,E1 -16398.463,E2 -16398.463} C_VEL
LIN {X 0,Y 298.39,Z 526.749,A -85,B 0,C 180,E1 -16400.689,E2 -16400.689} C_VEL
LIN {X 0,Y 297.517,Z 530.557,A -85,B 0,C 180,E1 -16402.884,E2 -16402.884} C_VEL
LIN {X 0,Y 296.758,Z 533.837,A -85,B 0,C 180,E1 -16405.846,E2 -16405.846} C_VEL
LIN {X 0,Y 296.33,Z 535.153,A -85,B 0,C 180,E1 -16408.651,E2 -16408.651} C_VEL
LIN {X 0,Y 296.212,Z 534.778,A -85,B 0,C 180,E1 -16411.331,E2 -16411.331} C_VEL
LIN {X 0,Y 296.286,Z 532.974,A -85,B 0,C 180,E1 -16413.876,E2 -16413.876} C_VEL
LIN {X 0,Y 296.654,Z 529.773,A -85,B 0,C 180,E1 -16416.339,E2 -16416.339} C_VEL
LIN {X 0,Y 297.093,Z 525.359,A -85,B 0,C 180,E1 -16418.677,E2 -16418.677} C_VEL
LIN {X 0,Y 297.717,Z 519.62,A -85,B 0,C 180,E1 -16420.937,E2 -16420.937} C_VEL
LIN {X 0,Y 298.553,Z 512.429,A -85,B 0,C 180,E1 -16423.132,E2 -16423.132} C_VEL
LIN {X 0,Y 299.461,Z 504.72,A -85,B 0,C 180,E1 -16425.024,E2 -16425.024} C_VEL
LIN {X 0,Y 300.747,Z 495.015,A -85,B 0,C 180,E1 -16426.932,E2 -16426.932} C_VEL
LIN {X 0,Y 302.014,Z 484.31,A -85,B 0,C 180,E1 -16428.631,E2 -16428.631} C_VEL
LIN {X 0,Y 303.366,Z 472.373,A -85,B 0,C 180,E1 -16430.12,E2 -16430.12} C_VEL
LIN {X 0,Y 304.127,Z 464.07,A -85,B 0,C 180,E1 -16430.968,E2 -16430.968} C_VEL
LIN {X 0,Y 302.415,Z 452.377,A -85,B 0,C 180,E1 -16432.068,E2 -16432.068} C_VEL
LIN {X 0,Y 300.059,Z 439.207,A -85,B 0,C 180,E1 -16433.059,E2 -16433.059} C_VEL
LIN {X 0,Y 297.872,Z 428.301,A -85,B 0,C 180,E1 -16433.704,E2 -16433.704} C_VEL
LIN {X 0,Y 298.189,Z 422.393,A -85,B 0,C 180,E1 -16437.172,E2 -16437.172} C_VEL
LIN {X 0,Y 298.553,Z 415.469,A -85,B 0,C 180,E1 -16441.257,E2 -16441.257} C_VEL
LIN {X 0,Y 299.007,Z 407.968,A -85,B 0,C 180,E1 -16445.709,E2 -16445.709} C_VEL
LIN {X 0,Y 298.789,Z 404.374,A -85,B 0,C 180,E1 -16447.89,E2 -16447.89} C_VEL
LIN {X 0,Y 298.567,Z 403.297,A -85,B 0,C 180,E1 -16448.599,E2 -16448.599} C_VEL
LIN {X 0,Y 298.54,Z 403.3,A -85,B 0,C 180,E1 -16452.177,E2 -16452.177} C_VEL
LIN {X 0,Y 298.596,Z 403.292,A -85,B 0,C 180,E1 -16454.992,E2 -16454.992} C_VEL
LIN {X 0,Y 298.592,Z 403.292,A -85,B 0,C 180,E1 -16459.144,E2 -16459.144} C_VEL
LIN {X 0,Y 298.713,Z 403.278,A -85,B 0,C 180,E1 -16461.882,E2 -16461.882} C_VEL
LIN {X 0,Y 298.618,Z 403.294,A -85,B 0,C 180,E1 -16465.272,E2 -16465.272} C_VEL
LIN {X 0,Y 298.635,Z 403.639,A -85,B 0,C 180,E1 -16465.949,E2 -16465.949} C_VEL
LIN {X 0,Y 299.455,Z 406.774,A -85,B 0,C 180,E1 -16468.652,E2 -16468.652} C_VEL
LIN {X 0,Y 299.172,Z 410.183,A -85,B 0,C 180,E1 -16471.343,E2 -16471.343} C_VEL
LIN {X 0,Y 298.486,Z 417.208,A -85,B 0,C 180,E1 -16476.758,E2 -16476.758} C_VEL
LIN {X 0,Y 297.911,Z 422.761,A -85,B 0,C 180,E1 -16480.875,E2 -16480.875} C_VEL
LIN {X 0,Y 297.653,Z 426.437,A -85,B 0,C 180,E1 -16483.567,E2 -16483.567} C_VEL
LIN {X 0,Y 300.399,Z 439.557,A -85,B 0,C 180,E1 -16484.47,E2 -16484.47} C_VEL
LIN {X 0,Y 302.266,Z 450.76,A -85,B 0,C 180,E1 -16485.478,E2 -16485.478} C_VEL
LIN {X 0,Y 303.13,Z 458.485,A -85,B 0,C 180,E1 -16486.323,E2 -16486.323} C_VEL
LIN {X 0,Y 301.981,Z 468.993,A -85,B 0,C 180,E1 -16487.607,E2 -16487.607} C_VEL
LIN {X 0,Y 300.89,Z 478.438,A -85,B 0,C 180,E1 -16489.083,E2 -16489.083} C_VEL
LIN {X 0,Y 299.954,Z 486.051,A -85,B 0,C 180,E1 -16490.573,E2 -16490.573} C_VEL
LIN {X 0,Y 298.994,Z 493.518,A -85,B 0,C 180,E1 -16492.394,E2 -16492.394} C_VEL
LIN {X 0,Y 298.168,Z 499.814,A -85,B 0,C 180,E1 -16494.357,E2 -16494.357} C_VEL
LIN {X 0,Y 297.56,Z 504.309,A -85,B 0,C 180,E1 -16496.168,E2 -16496.168} C_VEL
LIN {X 0,Y 297.088,Z 508.136,A -85,B 0,C 180,E1 -16498.233,E2 -16498.233} C_VEL
LIN {X 0,Y 296.84,Z 510.185,A -85,B 0,C 180,E1 -16499.81,E2 -16499.81} C_VEL
LIN {X 0,Y 296.659,Z 511.623,A -85,B 0,C 180,E1 -16501.477,E2 -16501.477} C_VEL
LIN {X 0,Y 296.627,Z 512.313,A -85,B 0,C 180,E1 -16503.016,E2 -16503.016} C_VEL
LIN {X 0,Y 296.713,Z 512.37,A -85,B 0,C 180,E1 -16504.639,E2 -16504.639} C_VEL
LIN {X 0,Y 296.94,Z 511.633,A -85,B 0,C 180,E1 -16506.418,E2 -16506.418} C_VEL
LIN {X 0,Y 297.461,Z 509.362,A -85,B 0,C 180,E1 -16508.77,E2 -16508.77} C_VEL
LIN {X 0,Y 298.258,Z 505.676,A -85,B 0,C 180,E1 -16511.06,E2 -16511.06} C_VEL
LIN {X 0,Y 299.227,Z 500.515,A -85,B 0,C 180,E1 -16513.273,E2 -16513.273} C_VEL
LIN {X 0,Y 300.258,Z 495.092,A -85,B 0,C 180,E1 -16515.043,E2 -16515.043} C_VEL
LIN {X 0,Y 301.416,Z 488.411,A -85,B 0,C 180,E1 -16516.767,E2 -16516.767} C_VEL
LIN {X 0,Y 302.915,Z 480.285,A -85,B 0,C 180,E1 -16518.432,E2 -16518.432} C_VEL
LIN {X 0,Y 304.374,Z 471.295,A -85,B 0,C 180,E1 -16519.888,E2 -16519.888} C_VEL
LIN {X 0,Y 305.678,Z 461.103,A -85,B 0,C 180,E1 -16521.208,E2 -16521.208} C_VEL
LIN {X 0,Y 304.546,Z 452.22,A -85,B 0,C 180,E1 -16522.295,E2 -16522.295} C_VEL
LIN {X 0,Y 302.186,Z 440.854,A -85,B 0,C 180,E1 -16523.491,E2 -16523.491} C_VEL
LIN {X 0,Y 299.169,Z 430.295,A -85,B 0,C 180,E1 -16524.435,E2 -16524.435} C_VEL
LIN {X 0,Y 298.408,Z 427.579,A -85,B 0,C 180,E1 -16524.672,E2 -16524.672} C_VEL
LIN {X 0,Y 298.694,Z 423.58,A -85,B 0,C 180,E1 -16527.884,E2 -16527.884} C_VEL
LIN {X 0,Y 299.206,Z 418.604,A -85,B 0,C 180,E1 -16531.981,E2 -16531.981} C_VEL
LIN {X 0,Y 299.511,Z 416.783,A -85,B 0,C 180,E1 -16533.524,E2 -16533.524} C_VEL
LIN {X 0,Y 299.754,Z 413.352,A -85,B 0,C 180,E1 -16536.511,E2 -16536.511} C_VEL
LIN {X 0,Y 299.623,Z 410.985,A -85,B 0,C 180,E1 -16538.719,E2 -16538.719} C_VEL
LIN {X 0,Y 298.878,Z 409.999,A -85,B 0,C 180,E1 -16539.822,E2 -16539.822} C_VEL
LIN {X 0,Y 295.839,Z 408.841,A -85,B 0,C 180,E1 -16541.626,E2 -16541.626} C_VEL
LIN {X 0,Y 293.252,Z 407.994,A -85,B 0,C 180,E1 -16543.092,E2 -16543.092} C_VEL
LIN {X 0,Y 292.097,Z 407.179,A -85,B 0,C 180,E1 -16544.228,E2 -16544.228} C_VEL
LIN {X 0,Y 291.979,Z 406.845,A -85,B 0,C 180,E1 -16544.612,E2 -16544.612} C_VEL
LIN {X 0,Y 291.516,Z 404.175,A -85,B 0,C 180,E1 -16547.823,E2 -16547.823} C_VEL
LIN {X 0,Y 291.684,Z 404.152,A -85,B 0,C 180,E1 -16551.688,E2 -16551.688} C_VEL
LIN {X 0,Y 291.615,Z 404.161,A -85,B 0,C 180,E1 -16554.469,E2 -16554.469} C_VEL
LIN {X 0,Y 291.875,Z 404.124,A -85,B 0,C 180,E1 -16558.621,E2 -16558.621} C_VEL
LIN {X 0,Y 291.875,Z 404.124,A -85,B 0,C 180,E1 -16561.38,E2 -16561.38} C_VEL
LIN {X 0,Y 291.615,Z 404.161,A -85,B 0,C 180,E1 -16565.532,E2 -16565.532} C_VEL
LIN {X 0,Y 291.688,Z 404.153,A -85,B 0,C 180,E1 -16568.313,E2 -16568.313} C_VEL
LIN {X 0,Y 291.502,Z 404.168,A -85,B 0,C 180,E1 -16572.533,E2 -16572.533} C_VEL
LIN {X 0,Y 291.535,Z 404.164,A -85,B 0,C 180,E1 -16575.378,E2 -16575.378} C_VEL
LIN {X 0,Y 291.464,Z 404.181,A -85,B 0,C 180,E1 -16579.895,E2 -16579.895} C_VEL
LIN {X 0,Y 291.408,Z 404.18,A -85,B 0,C 180,E1 -16584.205,E2 -16584.205} C_VEL
LIN {X 0,Y 291.405,Z 404.18,A -85,B 0,C 180,E1 -16587.274,E2 -16587.274} C_VEL
LIN {X 0,Y 291.32,Z 404.193,A -85,B 0,C 180,E1 -16590.439,E2 -16590.439} C_VEL
LIN {X 0,Y 291.328,Z 404.197,A -85,B 0,C 180,E1 -16593.701,E2 -16593.701} C_VEL
LIN {X 0,Y 291.389,Z 404.19,A -85,B 0,C 180,E1 -16597.264,E2 -16597.264} C_VEL
LIN {X 0,Y 291.416,Z 404.307,A -85,B 0,C 180,E1 -16599.836,E2 -16599.836} C_VEL
LIN {X 0,Y 292.426,Z 409.07,A -85,B 0,C 180,E1 -16604.185,E2 -16604.185} C_VEL
LIN {X 0,Y 293.383,Z 413.779,A -85,B 0,C 180,E1 -16607.954,E2 -16607.954} C_VEL
LIN {X 0,Y 294.316,Z 418.871,A -85,B 0,C 180,E1 -16611.626,E2 -16611.626} C_VEL
LIN {X 0,Y 295.358,Z 424.253,A -85,B 0,C 180,E1 -16615.179,E2 -16615.179} C_VEL
LIN {X 0,Y 295.823,Z 428.427,A -85,B 0,C 180,E1 -16617.692,E2 -16617.692} C_VEL
LIN {X 0,Y 294.227,Z 435.509,A -85,B 0,C 180,E1 -16621.467,E2 -16621.467} C_VEL
LIN {X 0,Y 292.904,Z 442.474,A -85,B 0,C 180,E1 -16624.993,E2 -16624.993} C_VEL
LIN {X 0,Y 295.782,Z 455.472,A -85,B 0,C 180,E1 -16625.87,E2 -16625.87} C_VEL
LIN {X 0,Y 297.502,Z 466.926,A -85,B 0,C 180,E1 -16626.822,E2 -16626.822} C_VEL
LIN {X 0,Y 298.363,Z 479.247,A -85,B 0,C 180,E1 -16628.045,E2 -16628.045} C_VEL
LIN {X 0,Y 298.169,Z 488.48,A -85,B 0,C 180,E1 -16629.118,E2 -16629.118} C_VEL
LIN {X 0,Y 296.472,Z 498.562,A -85,B 0,C 180,E1 -16630.441,E2 -16630.441} C_VEL
LIN {X 0,Y 294.829,Z 507.771,A -85,B 0,C 180,E1 -16631.951,E2 -16631.951} C_VEL
LIN {X 0,Y 293.507,Z 516.128,A -85,B 0,C 180,E1 -16633.663,E2 -16633.663} C_VEL
LIN {X 0,Y 292.113,Z 524.276,A -85,B 0,C 180,E1 -16635.727,E2 -16635.727} C_VEL
LIN {X 0,Y 291.054,Z 529.78,A -85,B 0,C 180,E1 -16637.452,E2 -16637.452} C_VEL
LIN {X 0,Y 290.293,Z 535.145,A -85,B 0,C 180,E1 -16639.542,E2 -16639.542} C_VEL
LIN {X 0,Y 289.521,Z 543.877,A -85,B 0,C 180,E1 -16643.732,E2 -16643.732} C_VEL
LIN {X 0,Y 289.458,Z 547.063,A -85,B 0,C 180,E1 -16645.826,E2 -16645.826} C_VEL
LIN {X 0,Y 289.492,Z 548.627,A -85,B 0,C 180,E1 -16647.22,E2 -16647.22} C_VEL
LIN {X 0,Y 289.465,Z 549.731,A -85,B 0,C 180,E1 -16648.612,E2 -16648.612} C_VEL
LIN {X 0,Y 289.467,Z 550.393,A -85,B 0,C 180,E1 -16650.003,E2 -16650.003} C_VEL
LIN {X 0,Y 289.457,Z 550.654,A -85,B 0,C 180,E1 -16651.394,E2 -16651.394} C_VEL
LIN {X 0,Y 289.492,Z 550.512,A -85,B 0,C 180,E1 -16652.786,E2 -16652.786} C_VEL
LIN {X 0,Y 289.462,Z 549.028,A -85,B 0,C 180,E1 -16655.456,E2 -16655.456} C_VEL
LIN {X 0,Y 289.641,Z 547.536,A -85,B 0,C 180,E1 -16656.971,E2 -16656.971} C_VEL
LIN {X 0,Y 290.083,Z 544.626,A -85,B 0,C 180,E1 -16659.064,E2 -16659.064} C_VEL
LIN {X 0,Y 290.79,Z 540.693,A -85,B 0,C 180,E1 -16661.151,E2 -16661.151} C_VEL
LIN {X 0,Y 291.808,Z 535.635,A -85,B 0,C 180,E1 -16663.229,E2 -16663.229} C_VEL
LIN {X 0,Y 293.316,Z 529.348,A -85,B 0,C 180,E1 -16665.285,E2 -16665.285} C_VEL
LIN {X 0,Y 294.839,Z 522.531,A -85,B 0,C 180,E1 -16667.098,E2 -16667.098} C_VEL
LIN {X 0,Y 296.317,Z 515.423,A -85,B 0,C 180,E1 -16668.677,E2 -16668.677} C_VEL
LIN {X 0,Y 298.54,Z 505.25,A -85,B 0,C 180,E1 -16670.501,E2 -16670.501} C_VEL
LIN {X 0,Y 300.996,Z 493.809,A -85,B 0,C 180,E1 -16672.12,E2 -16672.12} C_VEL
LIN {X 0,Y 301.868,Z 487.051,A -85,B 0,C 180,E1 -16672.955,E2 -16672.955} C_VEL
LIN {X 0,Y 301.934,Z 478.169,A -85,B 0,C 180,E1 -16674.015,E2 -16674.015} C_VEL
LIN {X 0,Y 301.201,Z 466.523,A -85,B 0,C 180,E1 -16675.25,E2 -16675.25} C_VEL
LIN {X 0,Y 299.212,Z 453.704,A -85,B 0,C 180,E1 -16676.488,E2 -16676.488} C_VEL
LIN {X 0,Y 295.922,Z 440.216,A -85,B 0,C 180,E1 -16677.689,E2 -16677.689} C_VEL
LIN {X 0,Y 294.282,Z 435.251,A -85,B 0,C 180,E1 -16678.166,E2 -16678.166} C_VEL
LIN {X 0,Y 294.222,Z 429.356,A -85,B 0,C 180,E1 -16679.715,E2 -16679.715} C_VEL
LIN {X 0,Y 294.943,Z 425.59,A -85,B 0,C 180,E1 -16681.619,E2 -16681.619} C_VEL
LIN {X 0,Y 294.871,Z 422.518,A -85,B 0,C 180,E1 -16683.245,E2 -16683.245} C_VEL
LIN {X 0,Y 293.7,Z 416.357,A -85,B 0,C 180,E1 -16686.746,E2 -16686.746} C_VEL
LIN {X 0,Y 292.508,Z 410.167,A -85,B 0,C 180,E1 -16690.448,E2 -16690.448} C_VEL
LIN {X 0,Y 291.35,Z 404.194,A -85,B 0,C 180,E1 -16694.298,E2 -16694.298} C_VEL
LIN {X 0,Y 291.303,Z 404.193,A -85,B 0,C 180,E1 -16698.413,E2 -16698.413} C_VEL
LIN {X 0,Y 291.343,Z 404.189,A -85,B 0,C 180,E1 -16701.156,E2 -16701.156} C_VEL
LIN {X 0,Y 291.364,Z 404.191,A -85,B 0,C 180,E1 -16704.626,E2 -16704.626} C_VEL
LIN {X 0,Y 291.374,Z 404.192,A -85,B 0,C 180,E1 -16707.95,E2 -16707.95} C_VEL
LIN {X 0,Y 291.33,Z 404.198,A -85,B 0,C 180,E1 -16711.152,E2 -16711.152} C_VEL
LIN {X 0,Y 291.35,Z 404.194,A -85,B 0,C 180,E1 -16714.265,E2 -16714.265} C_VEL
LIN {X 0,Y 291.361,Z 404.192,A -85,B 0,C 180,E1 -16717.297,E2 -16717.297} C_VEL
LIN {X 0,Y 291.468,Z 404.179,A -85,B 0,C 180,E1 -16720.27,E2 -16720.27} C_VEL
LIN {X 0,Y 291.525,Z 404.273,A -85,B 0,C 180,E1 -16723.184,E2 -16723.184} C_VEL
LIN {X 0,Y 292.298,Z 407.314,A -85,B 0,C 180,E1 -16726.087,E2 -16726.087} C_VEL
LIN {X 0,Y 293.426,Z 412.327,A -85,B 0,C 180,E1 -16730.348,E2 -16730.348} C_VEL
LIN {X 0,Y 294.101,Z 415.845,A -85,B 0,C 180,E1 -16733.137,E2 -16733.137} C_VEL
LIN {X 0,Y 294.317,Z 419.623,A -85,B 0,C 180,E1 -16735.892,E2 -16735.892} C_VEL
LIN {X 0,Y 293.797,Z 423.717,A -85,B 0,C 180,E1 -16738.629,E2 -16738.629} C_VEL
LIN {X 0,Y 292.936,Z 430.025,A -85,B 0,C 180,E1 -16742.707,E2 -16742.707} C_VEL
LIN {X 0,Y 294.207,Z 433.443,A -85,B 0,C 180,E1 -16743.101,E2 -16743.101} C_VEL
LIN {X 0,Y 298.458,Z 444.872,A -85,B 0,C 180,E1 -16744.473,E2 -16744.473} C_VEL
LIN {X 0,Y 301.359,Z 455.759,A -85,B 0,C 180,E1 -16745.794,E2 -16745.794} C_VEL
LIN {X 0,Y 303.281,Z 467.752,A -85,B 0,C 180,E1 -16747.322,E2 -16747.322} C_VEL
LIN {X 0,Y 303.573,Z 472.779,A -85,B 0,C 180,E1 -16747.984,E2 -16747.984} C_VEL
LIN {X 0,Y 301.476,Z 484.069,A -85,B 0,C 180,E1 -16749.391,E2 -16749.391} C_VEL
LIN {X 0,Y 299.337,Z 494.356,A -85,B 0,C 180,E1 -16750.997,E2 -16750.997} C_VEL
LIN {X 0,Y 297.04,Z 504.382,A -85,B 0,C 180,E1 -16752.974,E2 -16752.974} C_VEL
LIN {X 0,Y 295.219,Z 511.968,A -85,B 0,C 180,E1 -16754.827,E2 -16754.827} C_VEL
LIN {X 0,Y 293.616,Z 518.428,A -85,B 0,C 180,E1 -16756.77,E2 -16756.77} C_VEL
LIN {X 0,Y 292.238,Z 524.134,A -85,B 0,C 180,E1 -16758.945,E2 -16758.945} C_VEL
LIN {X 0,Y 291.043,Z 528.742,A -85,B 0,C 180,E1 -16761.236,E2 -16761.236} C_VEL
LIN {X 0,Y 290.379,Z 531.554,A -85,B 0,C 180,E1 -16763.112,E2 -16763.112} C_VEL
LIN {X 0,Y 289.655,Z 534.294,A -85,B 0,C 180,E1 -16765.896,E2 -16765.896} C_VEL
LIN {X 0,Y 289.369,Z 535.106,A -85,B 0,C 180,E1 -16767.481,E2 -16767.481} C_VEL
LIN {X 0,Y 289.193,Z 535.408,A -85,B 0,C 180,E1 -16769.08,E2 -16769.08} C_VEL
LIN {X 0,Y 289.099,Z 534.747,A -85,B 0,C 180,E1 -16771.692,E2 -16771.692} C_VEL
LIN {X 0,Y 289.23,Z 532.635,A -85,B 0,C 180,E1 -16774.29,E2 -16774.29} C_VEL
LIN {X 0,Y 289.652,Z 529.204,A -85,B 0,C 180,E1 -16776.8,E2 -16776.8} C_VEL
LIN {X 0,Y 290.113,Z 524.511,A -85,B 0,C 180,E1 -16779.173,E2 -16779.173} C_VEL
LIN {X 0,Y 290.795,Z 518.497,A -85,B 0,C 180,E1 -16781.475,E2 -16781.475} C_VEL
LIN {X 0,Y 291.69,Z 511.04,A -85,B 0,C 180,E1 -16783.709,E2 -16783.709} C_VEL
LIN {X 0,Y 292.87,Z 501.745,A -85,B 0,C 180,E1 -16785.897,E2 -16785.897} C_VEL
LIN {X 0,Y 294.022,Z 493.011,A -85,B 0,C 180,E1 -16787.561,E2 -16787.561} C_VEL
LIN {X 0,Y 295.271,Z 482.847,A -85,B 0,C 180,E1 -16789.137,E2 -16789.137} C_VEL
LIN {X 0,Y 296.534,Z 471.927,A -85,B 0,C 180,E1 -16790.504,E2 -16790.504} C_VEL
LIN {X 0,Y 297.147,Z 464.258,A -85,B 0,C 180,E1 -16791.306,E2 -16791.306} C_VEL
LIN {X 0,Y 295.232,Z 451.317,A -85,B 0,C 180,E1 -16792.537,E2 -16792.537} C_VEL
LIN {X 0,Y 292.701,Z 437.942,A -85,B 0,C 180,E1 -16793.537,E2 -16793.537} C_VEL
LIN {X 0,Y 290.814,Z 428.427,A -85,B 0,C 180,E1 -16794.121,E2 -16794.121} C_VEL
LIN {X 0,Y 291.206,Z 422.06,A -85,B 0,C 180,E1 -16797.928,E2 -16797.928} C_VEL
LIN {X 0,Y 291.501,Z 416.632,A -85,B 0,C 180,E1 -16801.168,E2 -16801.168} C_VEL
LIN {X 0,Y 291.898,Z 410.129,A -85,B 0,C 180,E1 -16805.078,E2 -16805.078} C_VEL
LIN {X 0,Y 291.913,Z 406.428,A -85,B 0,C 180,E1 -16807.34,E2 -16807.34} C_VEL
LIN {X 0,Y 291.533,Z 404.173,A -85,B 0,C 180,E1 -16808.798,E2 -16808.798} C_VEL
LIN {X 0,Y 291.489,Z 404.176,A -85,B 0,C 180,E1 -16813.18,E2 -16813.18} C_VEL
LIN {X 0,Y 291.524,Z 404.172,A -85,B 0,C 180,E1 -16816.047,E2 -16816.047} C_VEL
LIN {X 0,Y 291.573,Z 404.167,A -85,B 0,C 180,E1 -16820.283,E2 -16820.283} C_VEL
LIN {X 0,Y 291.698,Z 404.152,A -85,B 0,C 180,E1 -16823.078,E2 -16823.078} C_VEL
LIN {X 0,Y 291.606,Z 404.344,A -85,B 0,C 180,E1 -16825.505,E2 -16825.505} C_VEL
LIN {X 0,Y 292.451,Z 407.876,A -85,B 0,C 180,E1 -16828.62,E2 -16828.62} C_VEL
LIN {X 0,Y 292.141,Z 411.305,A -85,B 0,C 180,E1 -16831.375,E2 -16831.375} C_VEL
LIN {X 0,Y 291.428,Z 418.418,A -85,B 0,C 180,E1 -16836.922,E2 -16836.922} C_VEL
LIN {X 0,Y 290.828,Z 423.981,A -85,B 0,C 180,E1 -16841.143,E2 -16841.143} C_VEL
LIN {X 0,Y 290.636,Z 426.659,A -85,B 0,C 180,E1 -16843.144,E2 -16843.144} C_VEL
LIN {X 0,Y 293.158,Z 438.547,A -85,B 0,C 180,E1 -16843.956,E2 -16843.956} C_VEL
LIN {X 0,Y 295.157,Z 450.083,A -85,B 0,C 180,E1 -16845.004,E2 -16845.004} C_VEL
LIN {X 0,Y 296.249,Z 459.073,A -85,B 0,C 180,E1 -16846.005,E2 -16846.005} C_VEL
LIN {X 0,Y 295.2,Z 468.577,A -85,B 0,C 180,E1 -16847.184,E2 -16847.184} C_VEL
LIN {X 0,Y 293.935,Z 478.927,A -85,B 0,C 180,E1 -16848.828,E2 -16848.828} C_VEL
LIN {X 0,Y 292.824,Z 487.624,A -85,B 0,C 180,E1 -16850.606,E2 -16850.606} C_VEL
LIN {X 0,Y 291.947,Z 494.184,A -85,B 0,C 180,E1 -16852.277,E2 -16852.277} C_VEL
LIN {X 0,Y 291.121,Z 500.24,A -85,B 0,C 180,E1 -16854.226,E2 -16854.226} C_VEL
LIN {X 0,Y 290.41,Z 505.488,A -85,B 0,C 180,E1 -16856.44,E2 -16856.44} C_VEL
LIN {X 0,Y 290.02,Z 508.55,A -85,B 0,C 180,E1 -16858.195,E2 -16858.195} C_VEL
LIN {X 0,Y 289.866,Z 509.928,A -85,B 0,C 180,E1 -16859.21,E2 -16859.21} C_VEL
LIN {X 0,Y 289.646,Z 511.377,A -85,B 0,C 180,E1 -16860.629,E2 -16860.629} C_VEL
LIN {X 0,Y 289.544,Z 512.439,A -85,B 0,C 180,E1 -16862.271,E2 -16862.271} C_VEL
LIN {X 0,Y 289.612,Z 512.808,A -85,B 0,C 180,E1 -16864.405,E2 -16864.405} C_VEL
LIN {X 0,Y 289.946,Z 511.838,A -85,B 0,C 180,E1 -16866.881,E2 -16866.881} C_VEL
LIN {X 0,Y 290.564,Z 509.403,A -85,B 0,C 180,E1 -16869.286,E2 -16869.286} C_VEL
LIN {X 0,Y 291.369,Z 505.553,A -85,B 0,C 180,E1 -16871.606,E2 -16871.606} C_VEL
LIN {X 0,Y 292.475,Z 500.212,A -85,B 0,C 180,E1 -16873.873,E2 -16873.873} C_VEL
LIN {X 0,Y 293.885,Z 493.128,A -85,B 0,C 180,E1 -16876.092,E2 -16876.092} C_VEL
LIN {X 0,Y 295.366,Z 485.487,A -85,B 0,C 180,E1 -16877.927,E2 -16877.927} C_VEL
LIN {X 0,Y 296.856,Z 477.332,A -85,B 0,C 180,E1 -16879.487,E2 -16879.487} C_VEL
LIN {X 0,Y 298.424,Z 467.338,A -85,B 0,C 180,E1 -16880.995,E2 -16880.995} C_VEL
LIN {X 0,Y 298.988,Z 461.984,A -85,B 0,C 180,E1 -16881.683,E2 -16881.683} C_VEL
LIN {X 0,Y 297.867,Z 453.279,A -85,B 0,C 180,E1 -16882.8,E2 -16882.8} C_VEL
LIN {X 0,Y 295.464,Z 441.565,A -85,B 0,C 180,E1 -16884.082,E2 -16884.082} C_VEL
LIN {X 0,Y 292.179,Z 430.487,A -85,B 0,C 180,E1 -16885.133,E2 -16885.133} C_VEL
LIN {X 0,Y 291.45,Z 427.88,A -85,B 0,C 180,E1 -16885.351,E2 -16885.351} C_VEL
LIN {X 0,Y 291.694,Z 424.658,A -85,B 0,C 180,E1 -16887.991,E2 -16887.991} C_VEL
LIN {X 0,Y 292.376,Z 418.972,A -85,B 0,C 180,E1 -16892.825,E2 -16892.825} C_VEL
LIN {X 0,Y 292.718,Z 415.471,A -85,B 0,C 180,E1 -16895.911,E2 -16895.911} C_VEL
LIN {X 0,Y 292.684,Z 412.324,A -85,B 0,C 180,E1 -16898.889,E2 -16898.889} C_VEL
LIN {X 0,Y 292.34,Z 409.439,A -85,B 0,C 180,E1 -16901.789,E2 -16901.789} C_VEL
LIN {X 0,Y 291.979,Z 406.845,A -85,B 0,C 180,E1 -16904.612,E2 -16904.612} C_VEL
LIN {X 0,Y 291.192,Z 405.998,A -85,B 0,C 180,E1 -16905.747,E2 -16905.747} C_VEL
LIN {X 0,Y 288.132,Z 405.25,A -85,B 0,C 180,E1 -16907.606,E2 -16907.606} C_VEL
LIN {X 0,Y 285.637,Z 405.066,A -85,B 0,C 180,E1 -16909.124,E2 -16909.124} C_VEL
LIN {X 0,Y 284.649,Z 405.038,A -85,B 0,C 180,E1 -16910.304,E2 -16910.304} C_VEL
LIN {X 0,Y 284.61,Z 405.035,A -85,B 0,C 180,E1 -16910.703,E2 -16910.703} C_VEL
LIN {X 0,Y 284.677,Z 405.029,A -85,B 0,C 180,E1 -16912.91,E2 -16912.91} C_VEL
LIN {X 0,Y 284.739,Z 405.019,A -85,B 0,C 180,E1 -16917.171,E2 -16917.171} C_VEL
LIN {X 0,Y 284.929,Z 404.995,A -85,B 0,C 180,E1 -16920,E2 -16920} C_VEL
LIN {X 0,Y 284.739,Z 405.017,A -85,B 0,C 180,E1 -16922.83,E2 -16922.83} C_VEL
LIN {X 0,Y 284.678,Z 405.019,A -85,B 0,C 180,E1 -16927.091,E2 -16927.091} C_VEL
LIN {X 0,Y 284.546,Z 405.035,A -85,B 0,C 180,E1 -16929.957,E2 -16929.957} C_VEL
LIN {X 0,Y 284.462,Z 405.052,A -85,B 0,C 180,E1 -16934.304,E2 -16934.304} C_VEL
LIN {X 0,Y 284.408,Z 405.059,A -85,B 0,C 180,E1 -16937.25,E2 -16937.25} C_VEL
LIN {X 0,Y 284.401,Z 405.061,A -85,B 0,C 180,E1 -16940.241,E2 -16940.241} C_VEL
LIN {X 0,Y 284.366,Z 405.058,A -85,B 0,C 180,E1 -16943.884,E2 -16943.884} C_VEL
LIN {X 0,Y 284.379,Z 405.055,A -85,B 0,C 180,E1 -16947.176,E2 -16947.176} C_VEL
LIN {X 0,Y 284.278,Z 405.074,A -85,B 0,C 180,E1 -16951.277,E2 -16951.277} C_VEL
LIN {X 0,Y 284.346,Z 405.065,A -85,B 0,C 180,E1 -16955.357,E2 -16955.357} C_VEL
LIN {X 0,Y 284.34,Z 405.255,A -85,B 0,C 180,E1 -16958.617,E2 -16958.617} C_VEL
LIN {X 0,Y 285.163,Z 408.965,A -85,B 0,C 180,E1 -16962.329,E2 -16962.329} C_VEL
LIN {X 0,Y 285.946,Z 412.542,A -85,B 0,C 180,E1 -16965.461,E2 -16965.461} C_VEL
LIN {X 0,Y 286.889,Z 417.56,A -85,B 0,C 180,E1 -16969.413,E2 -16969.413} C_VEL
LIN {X 0,Y 287.991,Z 423.525,A -85,B 0,C 180,E1 -16973.642,E2 -16973.642} C_VEL
LIN {X 0,Y 288.822,Z 428.472,A -85,B 0,C 180,E1 -16976.809,E2 -16976.809} C_VEL
LIN {X 0,Y 288.855,Z 429.868,A -85,B 0,C 180,E1 -16977.642,E2 -16977.642} C_VEL
LIN {X 0,Y 286.877,Z 438.327,A -85,B 0,C 180,E1 -16982.264,E2 -16982.264} C_VEL
LIN {X 0,Y 286.123,Z 442.091,A -85,B 0,C 180,E1 -16984.255,E2 -16984.255} C_VEL
LIN {X 0,Y 289.087,Z 455.492,A -85,B 0,C 180,E1 -16985.221,E2 -16985.221} C_VEL
LIN {X 0,Y 290.922,Z 467.831,A -85,B 0,C 180,E1 -16986.301,E2 -16986.301} C_VEL
LIN {X 0,Y 291.678,Z 479.565,A -85,B 0,C 180,E1 -16987.515,E2 -16987.515} C_VEL
LIN {X 0,Y 291.526,Z 488.669,A -85,B 0,C 180,E1 -16988.619,E2 -16988.619} C_VEL
LIN {X 0,Y 289.79,Z 498.639,A -85,B 0,C 180,E1 -16989.971,E2 -16989.971} C_VEL
LIN {X 0,Y 288.066,Z 507.728,A -85,B 0,C 180,E1 -16991.512,E2 -16991.512} C_VEL
LIN {X 0,Y 286.661,Z 516.042,A -85,B 0,C 180,E1 -16993.269,E2 -16993.269} C_VEL
LIN {X 0,Y 285.217,Z 524.102,A -85,B 0,C 180,E1 -16995.374,E2 -16995.374} C_VEL
LIN {X 0,Y 284.108,Z 529.568,A -85,B 0,C 180,E1 -16997.14,E2 -16997.14} C_VEL
LIN {X 0,Y 283.257,Z 534.897,A -85,B 0,C 180,E1 -16999.279,E2 -16999.279} C_VEL
LIN {X 0,Y 282.466,Z 543.412,A -85,B 0,C 180,E1 -17003.575,E2 -17003.575} C_VEL
LIN {X 0,Y 282.361,Z 546.668,A -85,B 0,C 180,E1 -17005.721,E2 -17005.721} C_VEL
LIN {X 0,Y 282.418,Z 548.268,A -85,B 0,C 180,E1 -17007.15,E2 -17007.15} C_VEL
LIN {X 0,Y 282.386,Z 549.436,A -85,B 0,C 180,E1 -17008.577,E2 -17008.577} C_VEL
LIN {X 0,Y 282.385,Z 550.14,A -85,B 0,C 180,E1 -17010.003,E2 -17010.003} C_VEL
LIN {X 0,Y 282.379,Z 550.438,A -85,B 0,C 180,E1 -17011.429,E2 -17011.429} C_VEL
LIN {X 0,Y 282.395,Z 550.336,A -85,B 0,C 180,E1 -17012.856,E2 -17012.856} C_VEL
LIN {X 0,Y 282.355,Z 549.156,A -85,B 0,C 180,E1 -17015.357,E2 -17015.357} C_VEL
LIN {X 0,Y 282.581,Z 547.506,A -85,B 0,C 180,E1 -17017.146,E2 -17017.146} C_VEL
LIN {X 0,Y 283.059,Z 544.672,A -85,B 0,C 180,E1 -17019.29,E2 -17019.29} C_VEL
LIN {X 0,Y 283.818,Z 540.844,A -85,B 0,C 180,E1 -17021.429,E2 -17021.429} C_VEL
LIN {X 0,Y 284.905,Z 535.91,A -85,B 0,C 180,E1 -17023.556,E2 -17023.556} C_VEL
LIN {X 0,Y 286.484,Z 529.734,A -85,B 0,C 180,E1 -17025.658,E2 -17025.658} C_VEL
LIN {X 0,Y 288.051,Z 523.168,A -85,B 0,C 180,E1 -17027.479,E2 -17027.479} C_VEL
LIN {X 0,Y 289.637,Z 516.054,A -85,B 0,C 180,E1 -17029.124,E2 -17029.124} C_VEL
LIN {X 0,Y 291.964,Z 506.202,A -85,B 0,C 180,E1 -17030.984,E2 -17030.984} C_VEL
LIN {X 0,Y 294.536,Z 495.083,A -85,B 0,C 180,E1 -17032.632,E2 -17032.632} C_VEL
LIN {X 0,Y 295.505,Z 488.596,A -85,B 0,C 180,E1 -17033.479,E2 -17033.479} C_VEL
LIN {X 0,Y 295.713,Z 479.116,A -85,B 0,C 180,E1 -17034.66,E2 -17034.66} C_VEL
LIN {X 0,Y 295.026,Z 467.282,A -85,B 0,C 180,E1 -17035.985,E2 -17035.985} C_VEL
LIN {X 0,Y 293.155,Z 454.547,A -85,B 0,C 180,E1 -17037.292,E2 -17037.292} C_VEL
LIN {X 0,Y 290.351,Z 442.693,A -85,B 0,C 180,E1 -17038.421,E2 -17038.421} C_VEL
LIN {X 0,Y 287.846,Z 435.134,A -85,B 0,C 180,E1 -17039.233,E2 -17039.233} C_VEL
LIN {X 0,Y 287.922,Z 426.675,A -85,B 0,C 180,E1 -17041.664,E2 -17041.664} C_VEL
LIN {X 0,Y 287.92,Z 423.936,A -85,B 0,C 180,E1 -17043.151,E2 -17043.151} C_VEL
LIN {X 0,Y 286.676,Z 417.464,A -85,B 0,C 180,E1 -17046.917,E2 -17046.917} C_VEL
LIN {X 0,Y 285.645,Z 411.944,A -85,B 0,C 180,E1 -17050.294,E2 -17050.294} C_VEL
LIN {X 0,Y 284.465,Z 405.862,A -85,B 0,C 180,E1 -17054.235,E2 -17054.235} C_VEL
LIN {X 0,Y 284.256,Z 405.079,A -85,B 0,C 180,E1 -17054.85,E2 -17054.85} C_VEL
LIN {X 0,Y 284.248,Z 405.075,A -85,B 0,C 180,E1 -17058.119,E2 -17058.119} C_VEL
LIN {X 0,Y 284.323,Z 405.059,A -85,B 0,C 180,E1 -17062.281,E2 -17062.281} C_VEL
LIN {X 0,Y 284.316,Z 405.069,A -85,B 0,C 180,E1 -17065.351,E2 -17065.351} C_VEL
LIN {X 0,Y 284.287,Z 405.072,A -85,B 0,C 180,E1 -17068.724,E2 -17068.724} C_VEL
LIN {X 0,Y 284.273,Z 405.074,A -85,B 0,C 180,E1 -17071.983,E2 -17071.983} C_VEL
LIN {X 0,Y 284.301,Z 405.071,A -85,B 0,C 180,E1 -17076.161,E2 -17076.161} C_VEL
LIN {X 0,Y 284.409,Z 405.06,A -85,B 0,C 180,E1 -17080.582,E2 -17080.582} C_VEL
LIN {X 0,Y 284.446,Z 405.323,A -85,B 0,C 180,E1 -17081.264,E2 -17081.264} C_VEL
LIN {X 0,Y 285.213,Z 408.05,A -85,B 0,C 180,E1 -17084.273,E2 -17084.273} C_VEL
LIN {X 0,Y 285.935,Z 411.132,A -85,B 0,C 180,E1 -17087.219,E2 -17087.219} C_VEL
LIN {X 0,Y 286.676,Z 414.416,A -85,B 0,C 180,E1 -17090.118,E2 -17090.118} C_VEL
LIN {X 0,Y 287.338,Z 417.873,A -85,B 0,C 180,E1 -17092.975,E2 -17092.975} C_VEL
LIN {X 0,Y 287.524,Z 421.632,A -85,B 0,C 180,E1 -17095.794,E2 -17095.794} C_VEL
LIN {X 0,Y 286.962,Z 425.717,A -85,B 0,C 180,E1 -17098.596,E2 -17098.596} C_VEL
LIN {X 0,Y 286.219,Z 430.26,A -85,B 0,C 180,E1 -17101.626,E2 -17101.626} C_VEL
LIN {X 0,Y 287.513,Z 433.696,A -85,B 0,C 180,E1 -17102.034,E2 -17102.034} C_VEL
LIN {X 0,Y 291.463,Z 443.766,A -85,B 0,C 180,E1 -17103.348,E2 -17103.348} C_VEL
LIN {X 0,Y 294.749,Z 455.264,A -85,B 0,C 180,E1 -17104.841,E2 -17104.841} C_VEL
LIN {X 0,Y 296.67,Z 466.191,A -85,B 0,C 180,E1 -17106.29,E2 -17106.29} C_VEL
LIN {X 0,Y 297.315,Z 473.355,A -85,B 0,C 180,E1 -17107.299,E2 -17107.299} C_VEL
LIN {X 0,Y 294.99,Z 485.697,A -85,B 0,C 180,E1 -17108.908,E2 -17108.908} C_VEL
LIN {X 0,Y 292.603,Z 496.28,A -85,B 0,C 180,E1 -17110.655,E2 -17110.655} C_VEL
LIN {X 0,Y 290.338,Z 505.624,A -85,B 0,C 180,E1 -17112.583,E2 -17112.583} C_VEL
LIN {X 0,Y 288.456,Z 512.934,A -85,B 0,C 180,E1 -17114.461,E2 -17114.461} C_VEL
LIN {X 0,Y 286.447,Z 520.403,A -85,B 0,C 180,E1 -17116.883,E2 -17116.883} C_VEL
LIN {X 0,Y 284.871,Z 526.367,A -85,B 0,C 180,E1 -17119.411,E2 -17119.411} C_VEL
LIN {X 0,Y 283.721,Z 530.513,A -85,B 0,C 180,E1 -17121.811,E2 -17121.811} C_VEL
LIN {X 0,Y 283.222,Z 532.551,A -85,B 0,C 180,E1 -17123.392,E2 -17123.392} C_VEL
LIN {X 0,Y 282.753,Z 534.058,A -85,B 0,C 180,E1 -17124.995,E2 -17124.995} C_VEL
LIN {X 0,Y 282.429,Z 535.069,A -85,B 0,C 180,E1 -17126.609,E2 -17126.609} C_VEL
LIN {X 0,Y 282.086,Z 535.605,A -85,B 0,C 180,E1 -17129.304,E2 -17129.304} C_VEL
LIN {X 0,Y 281.997,Z 534.636,A -85,B 0,C 180,E1 -17132.071,E2 -17132.071} C_VEL
LIN {X 0,Y 282.198,Z 532.278,A -85,B 0,C 180,E1 -17134.726,E2 -17134.726} C_VEL
LIN {X 0,Y 282.644,Z 528.54,A -85,B 0,C 180,E1 -17137.277,E2 -17137.277} C_VEL
LIN {X 0,Y 283.134,Z 523.616,A -85,B 0,C 180,E1 -17139.689,E2 -17139.689} C_VEL
LIN {X 0,Y 283.893,Z 517.317,A -85,B 0,C 180,E1 -17142.037,E2 -17142.037} C_VEL
LIN {X 0,Y 284.871,Z 509.486,A -85,B 0,C 180,E1 -17144.317,E2 -17144.317} C_VEL
LIN {X 0,Y 286.016,Z 500.905,A -85,B 0,C 180,E1 -17146.321,E2 -17146.321} C_VEL
LIN {X 0,Y 287.357,Z 490.62,A -85,B 0,C 180,E1 -17148.24,E2 -17148.24} C_VEL
LIN {X 0,Y 288.68,Z 480.269,A -85,B 0,C 180,E1 -17149.803,E2 -17149.803} C_VEL
LIN {X 0,Y 290.028,Z 468.307,A -85,B 0,C 180,E1 -17151.232,E2 -17151.232} C_VEL
LIN {X 0,Y 290.105,Z 464.338,A -85,B 0,C 180,E1 -17151.653,E2 -17151.653} C_VEL
LIN {X 0,Y 288.235,Z 451.87,A -85,B 0,C 180,E1 -17152.878,E2 -17152.878} C_VEL
LIN {X 0,Y 285.874,Z 439.02,A -85,B 0,C 180,E1 -17153.881,E2 -17153.881} C_VEL
LIN {X 0,Y 283.809,Z 428.651,A -85,B 0,C 180,E1 -17154.504,E2 -17154.504} C_VEL
LIN {X 0,Y 284.165,Z 422.884,A -85,B 0,C 180,E1 -17157.986,E2 -17157.986} C_VEL
LIN {X 0,Y 284.546,Z 416.269,A -85,B 0,C 180,E1 -17162.01,E2 -17162.01} C_VEL
LIN {X 0,Y 284.963,Z 409.95,A -85,B 0,C 180,E1 -17165.856,E2 -17165.856} C_VEL
LIN {X 0,Y 284.681,Z 406.13,A -85,B 0,C 180,E1 -17168.262,E2 -17168.262} C_VEL
LIN {X 0,Y 284.48,Z 405.052,A -85,B 0,C 180,E1 -17169.006,E2 -17169.006} C_VEL
LIN {X 0,Y 284.429,Z 405.056,A -85,B 0,C 180,E1 -17172.749,E2 -17172.749} C_VEL
LIN {X 0,Y 284.484,Z 405.05,A -85,B 0,C 180,E1 -17175.694,E2 -17175.694} C_VEL
LIN {X 0,Y 284.518,Z 405.046,A -85,B 0,C 180,E1 -17180.04,E2 -17180.04} C_VEL
LIN {X 0,Y 284.653,Z 405.029,A -85,B 0,C 180,E1 -17182.906,E2 -17182.906} C_VEL
LIN {X 0,Y 284.578,Z 405.045,A -85,B 0,C 180,E1 -17185.038,E2 -17185.038} C_VEL
LIN {X 0,Y 285.443,Z 409.027,A -85,B 0,C 180,E1 -17188.586,E2 -17188.586} C_VEL
LIN {X 0,Y 285.108,Z 412.461,A -85,B 0,C 180,E1 -17191.409,E2 -17191.409} C_VEL
LIN {X 0,Y 284.48,Z 417.775,A -85,B 0,C 180,E1 -17195.668,E2 -17195.668} C_VEL
LIN {X 0,Y 284.134,Z 421.447,A -85,B 0,C 180,E1 -17198.531,E2 -17198.531} C_VEL
LIN {X 0,Y 283.609,Z 426.825,A -85,B 0,C 180,E1 -17202.656,E2 -17202.656} C_VEL
LIN {X 0,Y 286.081,Z 438.432,A -85,B 0,C 180,E1 -17203.493,E2 -17203.493} C_VEL
LIN {X 0,Y 288.025,Z 449.159,A -85,B 0,C 180,E1 -17204.48,E2 -17204.48} C_VEL
LIN {X 0,Y 289.374,Z 459.638,A -85,B 0,C 180,E1 -17205.672,E2 -17205.672} C_VEL
LIN {X 0,Y 288.172,Z 470.001,A -85,B 0,C 180,E1 -17207.014,E2 -17207.014} C_VEL
LIN {X 0,Y 286.99,Z 479.397,A -85,B 0,C 180,E1 -17208.56,E2 -17208.56} C_VEL
LIN {X 0,Y 285.79,Z 488.306,A -85,B 0,C 180,E1 -17210.434,E2 -17210.434} C_VEL
LIN {X 0,Y 284.736,Z 495.935,A -85,B 0,C 180,E1 -17212.49,E2 -17212.49} C_VEL
LIN {X 0,Y 283.996,Z 501.165,A -85,B 0,C 180,E1 -17214.279,E2 -17214.279} C_VEL
LIN {X 0,Y 283.294,Z 506.214,A -85,B 0,C 180,E1 -17216.518,E2 -17216.518} C_VEL
LIN {X 0,Y 282.944,Z 508.965,A -85,B 0,C 180,E1 -17218.156,E2 -17218.156} C_VEL
LIN {X 0,Y 282.686,Z 511.01,A -85,B 0,C 180,E1 -17219.812,E2 -17219.812} C_VEL
LIN {X 0,Y 282.457,Z 512.808,A -85,B 0,C 180,E1 -17222.224,E2 -17222.224} C_VEL
LIN {X 0,Y 282.572,Z 513.193,A -85,B 0,C 180,E1 -17224.888,E2 -17224.888} C_VEL
LIN {X 0,Y 282.955,Z 512.024,A -85,B 0,C 180,E1 -17227.363,E2 -17227.363} C_VEL
LIN {X 0,Y 283.674,Z 509.425,A -85,B 0,C 180,E1 -17229.824,E2 -17229.824} C_VEL
LIN {X 0,Y 284.554,Z 505.421,A -85,B 0,C 180,E1 -17232.188,E2 -17232.188} C_VEL
LIN {X 0,Y 285.764,Z 499.883,A -85,B 0,C 180,E1 -17234.503,E2 -17234.503} C_VEL
LIN {X 0,Y 286.921,Z 494.402,A -85,B 0,C 180,E1 -17236.263,E2 -17236.263} C_VEL
LIN {X 0,Y 288.318,Z 487.571,A -85,B 0,C 180,E1 -17238.021,E2 -17238.021} C_VEL
LIN {X 0,Y 289.898,Z 479.47,A -85,B 0,C 180,E1 -17239.674,E2 -17239.674} C_VEL
LIN {X 0,Y 291.509,Z 470.203,A -85,B 0,C 180,E1 -17241.184,E2 -17241.184} C_VEL
LIN {X 0,Y 292.385,Z 464.129,A -85,B 0,C 180,E1 -17241.999,E2 -17241.999} C_VEL
LIN {X 0,Y 291.274,Z 454.573,A -85,B 0,C 180,E1 -17243.289,E2 -17243.289} C_VEL
LIN {X 0,Y 289.061,Z 443.396,A -85,B 0,C 180,E1 -17244.593,E2 -17244.593} C_VEL
LIN {X 0,Y 285.928,Z 432.755,A -85,B 0,C 180,E1 -17245.682,E2 -17245.682} C_VEL
LIN {X 0,Y 284.518,Z 428.08,A -85,B 0,C 180,E1 -17246.13,E2 -17246.13} C_VEL
LIN {X 0,Y 284.974,Z 423.039,A -85,B 0,C 180,E1 -17250.447,E2 -17250.447} C_VEL
LIN {X 0,Y 285.489,Z 419.329,A -85,B 0,C 180,E1 -17253.698,E2 -17253.698} C_VEL
LIN {X 0,Y 285.789,Z 415.948,A -85,B 0,C 180,E1 -17256.83,E2 -17256.83} C_VEL
LIN {X 0,Y 285.684,Z 412.875,A -85,B 0,C 180,E1 -17259.855,E2 -17259.855} C_VEL
LIN {X 0,Y 285.124,Z 408.808,A -85,B 0,C 180,E1 -17264.268,E2 -17264.268} C_VEL
LIN {X 0,Y 284.498,Z 405.047,A -85,B 0,C 180,E1 -17268.873,E2 -17268.873} C_VEL
LIN {X 0,Y 284.61,Z 405.035,A -85,B 0,C 180,E1 -17270.703,E2 -17270.703} C_VEL
LIN {X 0,Y 284.013,Z 405.112,A -85,B 0,C 180,E1 -17271.884,E2 -17271.884} C_VEL
LIN {X 0,Y 281.076,Z 405.474,A -85,B 0,C 180,E1 -17273.804,E2 -17273.804} C_VEL
LIN {X 0,Y 278.613,Z 405.781,A -85,B 0,C 180,E1 -17275.365,E2 -17275.365} C_VEL
LIN {X 0,Y 277.677,Z 405.895,A -85,B 0,C 180,E1 -17276.577,E2 -17276.577} C_VEL
LIN {X 0,Y 277.669,Z 405.898,A -85,B 0,C 180,E1 -17276.986,E2 -17276.986} C_VEL
LIN {X 0,Y 277.886,Z 405.872,A -85,B 0,C 180,E1 -17280,E2 -17280} C_VEL
LIN {X 0,Y 277.694,Z 405.893,A -85,B 0,C 180,E1 -17282.902,E2 -17282.902} C_VEL
LIN {X 0,Y 277.633,Z 405.898,A -85,B 0,C 180,E1 -17287.272,E2 -17287.272} C_VEL
LIN {X 0,Y 277.486,Z 405.916,A -85,B 0,C 180,E1 -17290.213,E2 -17290.213} C_VEL
LIN {X 0,Y 277.415,Z 405.927,A -85,B 0,C 180,E1 -17294.676,E2 -17294.676} C_VEL
LIN {X 0,Y 277.352,Z 405.933,A -85,B 0,C 180,E1 -17299.234,E2 -17299.234} C_VEL
LIN {X 0,Y 277.325,Z 405.935,A -85,B 0,C 180,E1 -17303.921,E2 -17303.921} C_VEL
LIN {X 0,Y 277.308,Z 405.936,A -85,B 0,C 180,E1 -17307.508,E2 -17307.508} C_VEL
LIN {X 0,Y 277.255,Z 405.945,A -85,B 0,C 180,E1 -17310.484,E2 -17310.484} C_VEL
LIN {X 0,Y 277.238,Z 405.951,A -85,B 0,C 180,E1 -17313.898,E2 -17313.898} C_VEL
LIN {X 0,Y 277.287,Z 405.981,A -85,B 0,C 180,E1 -17317.018,E2 -17317.018} C_VEL
LIN {X 0,Y 278.064,Z 409.718,A -85,B 0,C 180,E1 -17321.083,E2 -17321.083} C_VEL
LIN {X 0,Y 279.025,Z 414.1,A -85,B 0,C 180,E1 -17325.156,E2 -17325.156} C_VEL
LIN {X 0,Y 279.894,Z 418.648,A -85,B 0,C 180,E1 -17328.877,E2 -17328.877} C_VEL
LIN {X 0,Y 280.948,Z 424.411,A -85,B 0,C 180,E1 -17333.109,E2 -17333.109} C_VEL
LIN {X 0,Y 281.89,Z 429.857,A -85,B 0,C 180,E1 -17336.741,E2 -17336.741} C_VEL
LIN {X 0,Y 281.664,Z 432.039,A -85,B 0,C 180,E1 -17338.034,E2 -17338.034} C_VEL
LIN {X 0,Y 279.827,Z 439.699,A -85,B 0,C 180,E1 -17342.318,E2 -17342.318} C_VEL
LIN {X 0,Y 279.37,Z 441.847,A -85,B 0,C 180,E1 -17343.478,E2 -17343.478} C_VEL
LIN {X 0,Y 282.527,Z 455.998,A -85,B 0,C 180,E1 -17344.569,E2 -17344.569} C_VEL
LIN {X 0,Y 284.319,Z 468.215,A -85,B 0,C 180,E1 -17345.698,E2 -17345.698} C_VEL
LIN {X 0,Y 285.038,Z 479.88,A -85,B 0,C 180,E1 -17346.961,E2 -17346.961} C_VEL
LIN {X 0,Y 284.89,Z 488.858,A -85,B 0,C 180,E1 -17348.096,E2 -17348.096} C_VEL
LIN {X 0,Y 283.123,Z 498.708,A -85,B 0,C 180,E1 -17349.478,E2 -17349.478} C_VEL
LIN {X 0,Y 281.341,Z 507.713,A -85,B 0,C 180,E1 -17351.054,E2 -17351.054} C_VEL
LIN {X 0,Y 279.851,Z 515.816,A -85,B 0,C 180,E1 -17352.81,E2 -17352.81} C_VEL
LIN {X 0,Y 278.329,Z 523.972,A -85,B 0,C 180,E1 -17355.004,E2 -17355.004} C_VEL
LIN {X 0,Y 277.179,Z 529.381,A -85,B 0,C 180,E1 -17356.813,E2 -17356.813} C_VEL
LIN {X 0,Y 276.237,Z 534.654,A -85,B 0,C 180,E1 -17359.003,E2 -17359.003} C_VEL
LIN {X 0,Y 275.327,Z 544.154,A -85,B 0,C 180,E1 -17364.143,E2 -17364.143} C_VEL
LIN {X 0,Y 275.272,Z 546.252,A -85,B 0,C 180,E1 -17365.611,E2 -17365.611} C_VEL
LIN {X 0,Y 275.322,Z 547.893,A -85,B 0,C 180,E1 -17367.077,E2 -17367.077} C_VEL
LIN {X 0,Y 275.31,Z 549.11,A -85,B 0,C 180,E1 -17368.541,E2 -17368.541} C_VEL
LIN {X 0,Y 275.306,Z 549.886,A -85,B 0,C 180,E1 -17370.003,E2 -17370.003} C_VEL
LIN {X 0,Y 275.302,Z 550.221,A -85,B 0,C 180,E1 -17371.466,E2 -17371.466} C_VEL
LIN {X 0,Y 275.3,Z 550.158,A -85,B 0,C 180,E1 -17372.93,E2 -17372.93} C_VEL
LIN {X 0,Y 275.259,Z 549.197,A -85,B 0,C 180,E1 -17375.272,E2 -17375.272} C_VEL
LIN {X 0,Y 275.516,Z 547.491,A -85,B 0,C 180,E1 -17377.331,E2 -17377.331} C_VEL
LIN {X 0,Y 276.023,Z 544.758,A -85,B 0,C 180,E1 -17379.529,E2 -17379.529} C_VEL
LIN {X 0,Y 276.859,Z 541.022,A -85,B 0,C 180,E1 -17381.72,E2 -17381.72} C_VEL
LIN {X 0,Y 278.018,Z 536.185,A -85,B 0,C 180,E1 -17383.898,E2 -17383.898} C_VEL
LIN {X 0,Y 279.984,Z 529.009,A -85,B 0,C 180,E1 -17386.406,E2 -17386.406} C_VEL
LIN {X 0,Y 281.615,Z 522.354,A -85,B 0,C 180,E1 -17388.279,E2 -17388.279} C_VEL
LIN {X 0,Y 283.847,Z 513.526,A -85,B 0,C 180,E1 -17390.285,E2 -17390.285} C_VEL
LIN {X 0,Y 286.406,Z 503.138,A -85,B 0,C 180,E1 -17392.168,E2 -17392.168} C_VEL
LIN {X 0,Y 288.849,Z 492.628,A -85,B 0,C 180,E1 -17393.672,E2 -17393.672} C_VEL
LIN {X 0,Y 289.499,Z 484.286,A -85,B 0,C 180,E1 -17394.801,E2 -17394.801} C_VEL
LIN {X 0,Y 289.264,Z 472.137,A -85,B 0,C 180,E1 -17396.297,E2 -17396.297} C_VEL
LIN {X 0,Y 287.978,Z 460.15,A -85,B 0,C 180,E1 -17397.628,E2 -17397.628} C_VEL
LIN {X 0,Y 285.332,Z 446.777,A -85,B 0,C 180,E1 -17399.026,E2 -17399.026} C_VEL
LIN {X 0,Y 281.604,Z 435.003,A -85,B 0,C 180,E1 -17400.359,E2 -17400.359} C_VEL
LIN {X 0,Y 281.675,Z 429.676,A -85,B 0,C 180,E1 -17401.969,E2 -17401.969} C_VEL
LIN {X 0,Y 281.15,Z 425.885,A -85,B 0,C 180,E1 -17403.366,E2 -17403.366} C_VEL
LIN {X 0,Y 280.283,Z 421.632,A -85,B 0,C 180,E1 -17405.223,E2 -17405.223} C_VEL
LIN {X 0,Y 278.837,Z 414.036,A -85,B 0,C 180,E1 -17409.906,E2 -17409.906} C_VEL
LIN {X 0,Y 277.638,Z 407.937,A -85,B 0,C 180,E1 -17413.943,E2 -17413.943} C_VEL
LIN {X 0,Y 277.211,Z 405.95,A -85,B 0,C 180,E1 -17415.483,E2 -17415.483} C_VEL
LIN {X 0,Y 277.205,Z 405.947,A -85,B 0,C 180,E1 -17419.52,E2 -17419.52} C_VEL
LIN {X 0,Y 277.269,Z 405.939,A -85,B 0,C 180,E1 -17422.53,E2 -17422.53} C_VEL
LIN {X 0,Y 277.255,Z 405.948,A -85,B 0,C 180,E1 -17426.105,E2 -17426.105} C_VEL
LIN {X 0,Y 277.237,Z 405.953,A -85,B 0,C 180,E1 -17429.535,E2 -17429.535} C_VEL
LIN {X 0,Y 277.262,Z 405.948,A -85,B 0,C 180,E1 -17432.853,E2 -17432.853} C_VEL
LIN {X 0,Y 277.264,Z 405.947,A -85,B 0,C 180,E1 -17436.073,E2 -17436.073} C_VEL
LIN {X 0,Y 277.308,Z 406.062,A -85,B 0,C 180,E1 -17438.439,E2 -17438.439} C_VEL
LIN {X 0,Y 277.879,Z 407.799,A -85,B 0,C 180,E1 -17440.804,E2 -17440.804} C_VEL
LIN {X 0,Y 278.587,Z 410.408,A -85,B 0,C 180,E1 -17443.888,E2 -17443.888} C_VEL
LIN {X 0,Y 279.24,Z 413.385,A -85,B 0,C 180,E1 -17446.908,E2 -17446.908} C_VEL
LIN {X 0,Y 279.935,Z 416.584,A -85,B 0,C 180,E1 -17449.878,E2 -17449.878} C_VEL
LIN {X 0,Y 280.571,Z 419.964,A -85,B 0,C 180,E1 -17452.805,E2 -17452.805} C_VEL
LIN {X 0,Y 280.777,Z 421.767,A -85,B 0,C 180,E1 -17454.253,E2 -17454.253} C_VEL
LIN {X 0,Y 280.495,Z 425.675,A -85,B 0,C 180,E1 -17457.127,E2 -17457.127} C_VEL
LIN {X 0,Y 279.671,Z 430.671,A -85,B 0,C 180,E1 -17460.449,E2 -17460.449} C_VEL
LIN {X 0,Y 280.963,Z 434.037,A -85,B 0,C 180,E1 -17460.893,E2 -17460.893} C_VEL
LIN {X 0,Y 285.555,Z 445.79,A -85,B 0,C 180,E1 -17462.558,E2 -17462.558} C_VEL
LIN {X 0,Y 288.476,Z 456.175,A -85,B 0,C 180,E1 -17463.998,E2 -17463.998} C_VEL
LIN {X 0,Y 290.43,Z 467.185,A -85,B 0,C 180,E1 -17465.554,E2 -17465.554} C_VEL
LIN {X 0,Y 291.056,Z 475.365,A -85,B 0,C 180,E1 -17466.76,E2 -17466.76} C_VEL
LIN {X 0,Y 288.815,Z 486.177,A -85,B 0,C 180,E1 -17468.219,E2 -17468.219} C_VEL
LIN {X 0,Y 286.433,Z 496.084,A -85,B 0,C 180,E1 -17469.889,E2 -17469.889} C_VEL
LIN {X 0,Y 284.099,Z 505.122,A -85,B 0,C 180,E1 -17471.776,E2 -17471.776} C_VEL
LIN {X 0,Y 282.098,Z 512.527,A -85,B 0,C 180,E1 -17473.675,E2 -17473.675} C_VEL
LIN {X 0,Y 280.337,Z 518.737,A -85,B 0,C 180,E1 -17475.634,E2 -17475.634} C_VEL
LIN {X 0,Y 278.893,Z 523.776,A -85,B 0,C 180,E1 -17477.601,E2 -17477.601} C_VEL
